	PERS robtarget H40:=[[108.33,-13.47,-153.24],[0.657572,-0.573127,-0.333582,0.357557],[-1,2,-3,0],[9E+09,-23.5,-50.1962,9E+09,9E+09,9E+09]];
	PERS robtarget H41:=[[106.78,-12.3,-180.44],[0.620126,-0.627649,-0.347001,0.317948],[-1,2,-3,0],[9E+09,-23.5,-50.1962,9E+09,9E+09,9E+09]];
	PERS robtarget H42:=[[107.29,-12.09,-209.23],[0.609617,-0.638486,-0.347041,0.316648],[-1,2,-3,0],[9E+09,-22,-50.1961,9E+09,9E+09,9E+09]];
	PERS robtarget H43:=[[151.42,1.00,-178.62],[0.641458,-0.319044,-0.596643,0.361609],[-1,1,-2,0],[9E+09,2.3391E-05,-89.9999,9E+09,9E+09,9E+09]];
	PERS robtarget H44:=[[151.41,-2.81,-181.55],[0.630186,-0.312225,-0.608538,0.367511],[-1,1,-2,0],[9E+09,-4.93563E-05,-90,9E+09,9E+09,9E+09]];
	PERS robtarget H45:=[[146.47,-4.42,-217.18],[0.639919,-0.321987,-0.598345,0.358905],[-1,1,-2,0],[9E+09,-7.78641E-06,-96,9E+09,9E+09,9E+09]];
	PERS robtarget H46:=[[145.71,-4.23,-254.81],[0.639921,-0.322004,-0.598339,0.358897],[-1,1,-2,0],[9E+09,-0.000496233,-90,9E+09,9E+09,9E+09]];
	PERS robtarget H47:=[[140.89,-9.14,-263.21],[0.710194,-0.342001,-0.385873,0.479337],[0,2,-3,0],[9E+09,7.53534E-05,-90.0001,9E+09,9E+09,9E+09]];
	PERS robtarget H48:=[[143.99,-1.12,-261.20],[0.728356,-0.371184,-0.349473,0.45781],[0,2,-3,0],[9E+09,-4.93563E-05,-90,9E+09,9E+09,9E+09]];
    PERS robtarget H49:=[[139.39,0.04,-263.43],[0.692369,-0.514594,-0.306839,0.402081],[0,3,-4,0],[9E+09,0.000594977,-90,9E+09,9E+09,9E+09]];

	PERS robtarget H50:=[[118.68,-79.14,-184.29],[0.585598,-0.475081,0.504836,-0.420137],[-1,1,-2,0],[9E+09,1.99993,81,9E+09,9E+09,9E+09]];
	PERS robtarget H51:=[[100.04,-72.41,-144.62],[0.366328,-0.602136,-0.49492,0.508222],[-1,-2,1,0],[9E+09,-5.97862,-90.0053,9E+09,9E+09,9E+09]];
	PERS robtarget H52:=[[102.34,-25.88,-157.75],[0.366327,-0.602138,-0.494919,0.508222],[-1,-2,1,0],[9E+09,-5.97862,-90.0053,9E+09,9E+09,9E+09]];
	PERS robtarget H53:=[[102.74,-20.19,-159.49],[0.422028,-0.65777,-0.448362,0.433824],[-1,-2,1,0],[9E+09,-5.9786,-90.0052,9E+09,9E+09,9E+09]];
	PERS robtarget H54:=[[120.26,-80.06,-182.83],[0.562619,-0.501182,0.519005,-0.403624],[-1,1,-2,0],[9E+09,3.00001,83.0001,9E+09,9E+09,9E+09]];
	PERS robtarget H55:=[[118.03,-29.06,-194.91],[0.620748,-0.499713,0.456833,-0.395302],[-1,1,-2,0],[9E+09,3.00001,82.9999,9E+09,9E+09,9E+09]];
	PERS robtarget H56:=[[100.61,-21.59,-159.10],[0.506741,-0.624171,-0.339688,0.488095],[-1,-1,1,0],[9E+09,2.59754E-05,-90.0022,9E+09,9E+09,9E+09]];
	PERS robtarget H57:=[[100.74,-23.77,-158.40],[0.460755,-0.573632,-0.396138,0.549296],[-1,-2,1,0],[9E+09,2.59754E-05,-90.0022,9E+09,9E+09,9E+09]];
	PERS robtarget H58:=[[100.20,-73.55,-145.24],[0.453285,-0.563309,-0.404643,0.559893],[-1,-2,1,0],[9E+09,-5.20202E-06,-90.0021,9E+09,9E+09,9E+09]];
    PERS robtarget H59:=[[111.03,-77.81,-189.53],[0.588099,-0.47989,0.482771,-0.436782],[-1,1,-2,0],[9E+09,3.00089,82.9986,9E+09,9E+09,9E+09]];

    PERS robtarget H98:=[[0,0,0],[0.73728,3.31828E-06,0.675588,2.33895E-06],[0,-1,0,0],[9E+09,9E+09,9E+09,9E+09,9E+09,9E+09]];
    PERS robtarget H99:=[[0,0,0],[0.73728,3.31828E-06,0.675588,2.33895E-06],[0,-1,0,0],[9E+09,9E+09,9E+09,9E+09,9E+09,9E+09]];

	PERS robtarget J1:=[[73.79,-16.15,-231.69],[0.592804,-0.401242,-0.200049,-0.669006],[-1,0,-2,0],[9E+09,20.3,-0.000874071,9E+09,9E+09,9E+09]];
	PERS robtarget J2:=[[83.36,-16.67,-232.23],[0.565018,-0.439497,-0.155442,-0.68076],[-1,0,-2,0],[9E+09,20.3,-0.000762002,9E+09,9E+09,9E+09]];
	PERS robtarget J3:=[[70.42,-14.81,-230.39],[0.645916,-0.288855,-0.284725,-0.646751],[-1,0,-2,0],[9E+09,20.3,-0.000874071,9E+09,9E+09,9E+09]];
	PERS robtarget J4:=[[0,-14.81,-230.39],[0.645916,-0.288853,-0.284725,-0.646752],[-1,0,-2,0],[9E+09,20.3,-0.000874071,9E+09,9E+09,9E+09]];
	PERS robtarget J5:=[[0,0,0],[0.73728,3.31828E-06,0.675588,2.33895E-06],[0,-1,0,0],[9E+09,9E+09,9E+09,9E+09,9E+09,9E+09]];

	PERS robtarget K1:=[[-87.2,-16.87,-232.73],[0.672861,-0.201577,-0.388086,-0.596669],[-1,0,-2,0],[9E+09,20.3,-0.000537865,9E+09,9E+09,9E+09]];
	PERS robtarget K2:=[[-95.39,-17.01,-232.66],[0.6898,-0.136714,-0.438311,-0.559793],[-1,0,-3,0],[9E+09,20.3,-0.000649933,9E+09,9E+09,9E+09]];
	PERS robtarget K3:=[[-77.34,-13.76,-231.53],[0.645912,-0.288853,-0.284724,-0.646757],[-1,0,-2,0],[9E+09,20.3,-0.000605106,9E+09,9E+09,9E+09]];
	PERS robtarget K4:=[[0,-13.76,-231.53],[0.645911,-0.288852,-0.284724,-0.646758],[-1,0,-2,0],[9E+09,20.3,-0.000649933,9E+09,9E+09,9E+09]];
	PERS robtarget K5:=[[0,0,0],[0.73728,3.31828E-06,0.675588,2.33895E-06],[0,-1,0,0],[9E+09,9E+09,9E+09,9E+09,9E+09,9E+09]];

	PERS robtarget L1:=[[0,0,0],[0.73728,3.31828E-06,0.675588,2.33895E-06],[0,-1,0,0],[9E+09,9E+09,9E+09,9E+09,9E+09,9E+09]];
	PERS robtarget L2:=[[0,0,0],[0.73728,3.31828E-06,0.675588,2.33895E-06],[0,-1,0,0],[9E+09,9E+09,9E+09,9E+09,9E+09,9E+09]];
	PERS robtarget L3:=[[0,0,0],[0.73728,3.31828E-06,0.675588,2.33895E-06],[0,-1,0,0],[9E+09,9E+09,9E+09,9E+09,9E+09,9E+09]];
	PERS robtarget L4:=[[0,0,0],[0.73728,3.31828E-06,0.675588,2.33895E-06],[0,-1,0,0],[9E+09,9E+09,9E+09,9E+09,9E+09,9E+09]];
    PERS robtarget L5:=[[0,0,0],[0.73728,3.31828E-06,0.675588,2.33895E-06],[0,-1,0,0],[9E+09,9E+09,9E+09,9E+09,9E+09,9E+09]];
    PERS robtarget L6:=[[0,0,0],[0.73728,3.31828E-06,0.675588,2.33895E-06],[0,-1,0,0],[9E+09,9E+09,9E+09,9E+09,9E+09,9E+09]];
    PERS robtarget L7:=[[0,0,0],[0.73728,3.31828E-06,0.675588,2.33895E-06],[0,-1,0,0],[9E+09,9E+09,9E+09,9E+09,9E+09,9E+09]];
    PERS robtarget L8:=[[0,0,0],[0.73728,3.31828E-06,0.675588,2.33895E-06],[0,-1,0,0],[9E+09,9E+09,9E+09,9E+09,9E+09,9E+09]];
    PERS robtarget L9:=[[0,0,0],[0.73728,3.31828E-06,0.675588,2.33895E-06],[0,-1,0,0],[9E+09,9E+09,9E+09,9E+09,9E+09,9E+09]];
    PERS robtarget L10:=[[0,0,0],[0.73728,3.31828E-06,0.675588,2.33895E-06],[0,-1,0,0],[9E+09,9E+09,9E+09,9E+09,9E+09,9E+09]];
    PERS robtarget L40:=[[0,-169.39,841.37],[0.442606,-0.811905,0.276598,-0.261544],[-1,1,-2,0],[9E+09,-14.1988,49.3012,9E+09,9E+09,9E+09]];
	PERS robtarget L41:=[[96.6934,-167.187,469.006],[0.634627,-0.665497,0.280508,-0.275094],[0,1,-2,0],[9E+09,-0.275255,46.2247,9E+09,9E+09,9E+09]];
	PERS robtarget L42:=[[96.95,-163.039,524.102],[0.613381,-0.680757,0.277205,-0.288948],[-1,1,-2,0],[9E+09,-3.95049,47.5495,9E+09,9E+09,9E+09]];
	PERS robtarget L43:=[[96.4403,0,0],[0.73728,3.31828E-06,0.675588,2.33895E-06],[0,-1,0,0],[9E+09,9E+09,9E+09,9E+09,9E+09,9E+09]];
	PERS robtarget L44:=[[96.4403,0,0],[0.73728,3.31828E-06,0.675588,2.33895E-06],[0,-1,0,0],[9E+09,9E+09,9E+09,9E+09,9E+09,9E+09]];
    PERS robtarget L45:=[[97.2063,-156.283,579.142],[0.580686,-0.706216,0.267929,-0.303771],[-1,1,-2,0],[9E+09,-8.10884,48.3912,9E+09,9E+09,9E+09]];
    PERS robtarget L46:=[[97.2552,-152.576,589.64],[0.574791,-0.71088,0.269371,-0.302828],[-1,1,-2,0],[9E+09,-8.96447,48.5355,9E+09,9E+09,9E+09]];
    PERS robtarget L47:=[[97.4579,-143.314,633.167],[0.544782,-0.734855,0.260153,-0.309065],[-1,1,-2,0],[9E+09,-12.438,49.062,9E+09,9E+09,9E+09]];
    PERS robtarget L48:=[[97.7028,-125.721,685.736],[0.505031,-0.765566,0.242802,-0.31607],[-1,1,-2,0],[9E+09,-16.8632,49.6368,9E+09,9E+09,9E+09]];
    PERS robtarget L49:=[[97.7897,-118.231,704.402],[0.49199,-0.775329,0.234663,-0.318974],[-1,1,-2,0],[9E+09,-18.2042,49.7958,9E+09,9E+09,9E+09]];
    PERS robtarget L50:=[[97.7897,-112.37,718.21],[0.610407,-0.715463,0.144537,-0.307611],[-1,1,-3,0],[9E+09,-18.2042,49.7958,9E+09,9E+09,9E+09]];

    PERS robtarget L40cramp1:=[[89.34,-171.59,828.86],[0.371994,-0.853426,0.291056,-0.220391],[-1,1,-2,0],[9E+09,-14.1988,49.3012,9E+09,9E+09,9E+09]];
    PERS robtarget L40cramp2:=[[89.66,-174.94,816.24],[0.319922,-0.878441,0.2998,-0.19003],[-1,1,-2,0],[9E+09,-14.1988,49.3012,9E+09,9E+09,9E+09]];


    PERS robtarget L68:=[[96.3294,-183.624,325.052],[0.732807,-0.547572,0.316136,-0.25143],[0,2,-3,0],[9E+09,11.563,48.937,9E+09,9E+09,9E+09]];
    PERS robtarget L69:=[[96.3488,-150.2,298.164],[0.659613,-0.633434,0.346072,-0.20954],[0,2,-2,0],[9E+09,9.82577,48.6742,9E+09,9E+09,9E+09]];
    PERS robtarget L67:=[[96.3401,-153.031,310.32],[0.720285,-0.563292,0.323715,-0.243106],[0,2,-3,0],[9E+09,8.96447,48.5355,9E+09,9E+09,9E+09]];
    PERS robtarget L66:=[[96.3373,-176.27,314.16],[0.672496,-0.593746,0.194944,-0.396502],[0,1,-3,0],[9E+09,11.0978,49.3364,9E+09,9E+09,9E+09]];
    PERS robtarget L65:=[[96.3969,-150.45,231.45],[0.672501,-0.59375,0.194937,-0.39649],[0,1,-2,0],[9E+09,15.8071,49.3364,9E+09,9E+09,9E+09]];
    PERS robtarget L64:=[[96.3969,-150.45,231.45],[0.672501,-0.59375,0.194937,-0.39649],[0,1,-2,0],[9E+09,15.8071,49.3364,9E+09,9E+09,9E+09]];
    PERS robtarget L63:=[[96.3115,-190.14,349.956],[0.72386,-0.558889,0.31987,-0.247696],[0,2,-3,0],[9E+09,9.82577,48.6742,9E+09,9E+09,9E+09]];
    PERS robtarget L62:=[[96.3013,-197.227,383.785],[0.712549,-0.57296,0.323832,-0.243152],[0,2,-3,0],[9E+09,7.68338,48.3166,9E+09,9E+09,9E+09]];
    PERS robtarget L61:=[[96.3326,-155.291,320.651],[0.74323,-0.532709,0.302829,-0.268562],[0,2,-3,0],[9E+09,8.10884,48.3912,9E+09,9E+09,9E+09]];
    PERS robtarget L60:=[[0,-199.67,711.03],[0.694049,-0.59574,0.215139,-0.342208],[-1,2,-3,0],[9E+09,-6.41779,48.0822,9E+09,9E+09,9E+09]];

	PERS robtarget M70:=[[-93.6428,-146.142,278.519],[0.617494,-0.211758,-0.675695,-0.342485],[-1,0,-2,0],[9E+09,9.82577,-48.6742,9E+09,9E+09,9E+09]];
	PERS robtarget L70:=[[96.3488,-145.531,278.717],[0.5807,-0.736812,0.322963,-0.124864],[0,2,-2,0],[9E+09,9.82577,48.6742,9E+09,9E+09,9E+09]];

    PERS robtarget M69:=[[-93.6428,-150.811,297.966],[0.566281,-0.122383,-0.698677,-0.419761],[-1,0,-2,0],[9E+09,9.82577,-48.6742,9E+09,9E+09,9E+09]];
    PERS robtarget M68:=[[-93.4449,-183.819,325.057],[0.649099,-0.0877175,-0.626165,-0.422957],[-1,0,-2,0],[9E+09,11.563,-48.937,9E+09,9E+09,9E+09]];
    PERS robtarget M67:=[[-93.5531,-153.581,310.245],[0.640867,-0.100792,-0.641818,-0.408901],[-1,0,-2,0],[9E+09,8.96447,-48.5355,9E+09,9E+09,9E+09]];
    PERS robtarget M66:=[[-93.5299,-177.55,313.42],[0.638045,-0.136384,-0.644614,-0.398463],[-1,0,-2,0],[9E+09,7.72271,-42.4887,9E+09,9E+09,9E+09]];
    PERS robtarget M65:=[[-94.1287,-400.46,231.46],[0.672498,-0.593754,0.194941,-0.396487],[0,1,-2,0],[9E+09,15.8062,49.3364,9E+09,9E+09,9E+09]];
    PERS robtarget M64:=[[-94.1287,-400.46,231.46],[0.672498,-0.593754,0.194941,-0.396487],[0,1,-2,0],[9E+09,15.8062,49.3364,9E+09,9E+09,9E+09]];
    PERS robtarget M63:=[[-93.2634,-190.289,349.9],[0.657211,-0.117717,-0.633101,-0.391663],[-1,0,-2,0],[9E+09,9.82577,-48.6742,9E+09,9E+09,9E+09]];
    PERS robtarget M62:=[[-93.0156,-197.372,383.803],[0.666771,-0.159333,-0.638564,-0.349665],[-1,0,-2,0],[9E+09,7.68338,-48.3166,9E+09,9E+09,9E+09]];
    PERS robtarget M61:=[[-93.4777,-155.55,320.558],[0.705794,-0.145598,-0.601393,-0.34494],[-1,0,-2,0],[9E+09,8.10884,-48.3912,9E+09,9E+09,9E+09]];
    PERS robtarget M60:=[[0,-199.66,711.57],[0.723621,-0.258575,-0.586981,-0.254884],[-1,0,-2,0],[9E+09,-6.41779,-48.0822,9E+09,9E+09,9E+09]];

	PERS robtarget M1:=[[0,0,0],[0.73728,3.31828E-06,0.675588,2.33895E-06],[0,-1,0,0],[9E+09,9E+09,9E+09,9E+09,9E+09,9E+09]];
	PERS robtarget M2:=[[0,0,0],[0.73728,3.31828E-06,0.675588,2.33895E-06],[0,-1,0,0],[9E+09,9E+09,9E+09,9E+09,9E+09,9E+09]];
	PERS robtarget M3:=[[0,0,0],[0.73728,3.31828E-06,0.675588,2.33895E-06],[0,-1,0,0],[9E+09,9E+09,9E+09,9E+09,9E+09,9E+09]];
	PERS robtarget M4:=[[0,0,0],[0.73728,3.31828E-06,0.675588,2.33895E-06],[0,-1,0,0],[9E+09,9E+09,9E+09,9E+09,9E+09,9E+09]];
    PERS robtarget M5:=[[0,0,0],[0.73728,3.31828E-06,0.675588,2.33895E-06],[0,-1,0,0],[9E+09,9E+09,9E+09,9E+09,9E+09,9E+09]];
    PERS robtarget M6:=[[0,0,0],[0.73728,3.31828E-06,0.675588,2.33895E-06],[0,-1,0,0],[9E+09,9E+09,9E+09,9E+09,9E+09,9E+09]];
    PERS robtarget M7:=[[0,0,0],[0.73728,3.31828E-06,0.675588,2.33895E-06],[0,-1,0,0],[9E+09,9E+09,9E+09,9E+09,9E+09,9E+09]];
    PERS robtarget M8:=[[0,0,0],[0.73728,3.31828E-06,0.675588,2.33895E-06],[0,-1,0,0],[9E+09,9E+09,9E+09,9E+09,9E+09,9E+09]];
    PERS robtarget M9:=[[0,0,0],[0.73728,3.31828E-06,0.675588,2.33895E-06],[0,-1,0,0],[9E+09,9E+09,9E+09,9E+09,9E+09,9E+09]];
    PERS robtarget M10:=[[111.15,-112.53,220.41],[0.643491,-0.632415,0.208259,-0.377624],[0,1,-2,0],[9E+09,10.5848,49.3365,9E+09,9E+09,9E+09]];
    PERS robtarget M40:=[[0,-168.58,841.23],[0.497618,-0.44465,-0.735594,-0.116468],[-1,0,-2,0],[9E+09,-14.1988,-49.3012,9E+09,9E+09,9E+09]];
	PERS robtarget M41:=[[-92.3859,-167.501,469.014],[0.646009,-0.277625,-0.665978,-0.249139],[-1,0,-2,0],[9E+09,-0.275255,-46.2247,9E+09,9E+09,9E+09]];
	PERS robtarget M42:=[[-92.0275,-163.382,524.16],[0.641706,-0.296382,-0.672629,-0.218956],[-1,0,-2,0],[9E+09,-3.95049,-47.5495,9E+09,9E+09,9E+09]];
	PERS robtarget M43:=[[-95.7201,0,0],[0.73728,3.31828E-06,0.675588,2.33895E-06],[0,-1,0,0],[9E+09,9E+09,9E+09,9E+09,9E+09,9E+09]];
	PERS robtarget M44:=[[-95.7201,0,0],[0.73728,3.31828E-06,0.675588,2.33895E-06],[0,-1,0,0],[9E+09,9E+09,9E+09,9E+09,9E+09,9E+09]];
    PERS robtarget M45:=[[-92.0423,-156.01,579.07],[0.629623,-0.325223,-0.681731,-0.181791],[-1,0,-2,0],[9E+09,-8.10884,-48.3912,9E+09,9E+09,9E+09]];
    PERS robtarget M46:=[[-92.0451,-152.729,589.619],[0.622938,-0.320879,-0.689165,-0.184493],[-1,0,-2,0],[9E+09,-8.96447,-48.5355,9E+09,9E+09,9E+09]];
    PERS robtarget M47:=[[-92.0568,-142.72,632.959],[0.608305,-0.355764,-0.693631,-0.149241],[-1,0,-2,0],[9E+09,-12.438,-49.062,9E+09,9E+09,9E+09]];
    PERS robtarget M48:=[[-92.0709,-124.754,685.369],[0.582927,-0.382483,-0.706223,-0.123094],[-1,0,-2,0],[9E+09,-16.8632,-49.6368,9E+09,9E+09,9E+09]];
    PERS robtarget M49:=[[-92.0759,-117.236,703.903],[0.574484,-0.388531,-0.710806,-0.117328],[-1,0,-2,0],[9E+09,-18.2042,-49.7958,9E+09,9E+09,9E+09]];
    PERS robtarget M50:=[[-92.0759,-111.375,717.71],[0.628488,-0.31192,-0.682674,-0.204122],[-1,0,-2,0],[9E+09,-18.2042,-49.7958,9E+09,9E+09,9E+09]];


!!!!!!!!!!!!!!!!!!!!!!END OF THE WRAPPER WELDS!!!!!!!!!!

	PERS robtarget AIRG50_1:=[[-520.73,-53.52,-86.29],[0.528398,-0.491715,0.591821,-0.358833],[-1,-3,2,0],[9E+09,-5.99999,96.0001,9E+09,9E+09,9E+09]];
	CONST robtarget AIRTOG40:=[[-143.55,-8.66,-258.80],[0.531165,-0.426072,0.558082,-0.474208],[-1,1,-2,0],[9E+09,4.25678,88.0425,9E+09,9E+09,9E+09]];
	CONST robtarget AIRTOG50:=[[-113.36,-82.97,-180.83],[0.229441,0.62405,-0.35786,-0.655634],[-1,-1,-3,0],[9E+09,2,-81,9E+09,9E+09,9E+09]];
	CONST robtarget AIRTOH50:=[[115.64,-84.86,-185.39],[0.583759,-0.477077,0.502947,-0.422693],[-1,1,-2,0],[9E+09,1.99998,81,9E+09,9E+09,9E+09]];
	CONST robtarget AIRTOH40:=[[147.28,-7.36,-258.56],[0.639947,-0.321989,-0.598323,0.35889],[-1,1,-2,0],[9E+09,0.0012601,-90,9E+09,9E+09,9E+09]];
	CONST robtarget AIRTOSNIFF_FRONT1:=[[-32.84,651.47,382.08],[0.458666,0.489208,0.507975,0.540615],[0,0,-2,1],[9E+09,0.00155109,179.999,9E+09,9E+09,9E+09]];
	CONST robtarget AIRTOSNIFF_FRONT2:=[[65.52,66.66,373.83],[0.458667,0.489243,0.508101,0.540464],[0,0,-2,1],[9E+09,0.00077165,180,9E+09,9E+09,9E+09]];
	CONST robtarget AIRTOSNIFF_BACK1:=[[30.52,-723.52,526.87],[0.502022,0.5218,-0.484293,-0.491081],[-1,-1,-2,1],[9E+09,0,0,9E+09,9E+09,9E+09]];


	CONST robtarget AIRTOU30_1:=[[288.8,655.25,389.82],[0.299157,-0.329043,-0.63518,0.631493],[-1,1,-2,0],[9E+09,-22,-135,9E+09,9E+09,9E+09]];
    CONST robtarget SPAGHAIR1:=[[10.28,-310.74,36.91],[0.687984,-0.0566141,-0.0392933,-0.722448],[0,-1,-1,0],[9E+09,0.000407913,0.000403513,9E+09,9E+09,9E+09]];
    CONST robtarget SPAGHAIR2:=[[6.27,-351.73,67.88],[0.547219,-0.440868,-0.452479,-0.549046],[-1,0,-2,0],[9E+09,0.000906752,0.000784547,9E+09,9E+09,9E+09]];
    CONST robtarget SPAGHAIR3:=[[-0.30,-21.47,198.76],[0.547881,-0.439991,-0.453355,-0.548365],[-1,0,-2,0],[9E+09,0.000927537,0.000829375,9E+09,9E+09,9E+09]];
    CONST robtarget SPAGHAIRp180:=[[0.12,-168.40,-471.89],[0.525941,0.414544,0.456451,-0.585828],[0,0,-4,0],[9E+09,-0.00069369,180,9E+09,9E+09,9E+09]];
    CONST robtarget AIRTOT30_1:=[[-387.74,-383.85,499.37],[0.413094,-0.652879,0.573252,-0.27292],[0,2,-3,0],[9E+09,-18.7937,76.4339,9E+09,9E+09,9E+09]];
    CONST robtarget AIRTOT30_2:=[[-149.56,-360.66,399.66],[0.413095,-0.652876,0.573254,-0.272923],[0,2,-2,0],[9E+09,-18.7937,76.4339,9E+09,9E+09,9E+09]];
    CONST robtarget AIRTOHSIDESEARCH_1:=[[336.07,-164.67,-442.68],[0.254905,-0.945405,0.203005,0.00489991],[-1,1,-1,0],[9E+09,0.000127316,-4.4762E-05,9E+09,9E+09,9E+09]];
    CONST robtarget AIRTOGSIDESEARCH_1:=[[-336.31,363.60,-301.34],[0.0476339,-0.197008,-0.979243,0.00193439],[-1,1,-1,0],[9E+09,0.0487537,179.953,9E+09,9E+09,9E+09]];

    CONST robtarget AIRTOU30_2:=[[-69.31,237.05,289.11],[0.401333,0.727401,-0.0339958,0.555577],[-1,0,-2,0],[9E+09,-22,-225,9E+09,9E+09,9E+09]];
    CONST robtarget AIRTOT30_3:=[[399.86,-369.93,558.91],[0.724495,0.0577651,-0.674607,0.129141],[-1,0,-2,0],[9E+09,-10.5388,-76.9656,9E+09,9E+09,9E+09]];
    CONST robtarget AIRTOAH118:=[[414.86,-318.11,504.4],[0.600973,-0.149246,-0.783454,-0.0525223],[-1,0,-2,0],[9E+09,-40,-74.7502,9E+09,9E+09,9E+09]];
    CONST robtarget AIRTOAG118:=[[-319.97,-306.98,657.22],[0.263609,-0.69609,0.660491,-0.098598],[-1,0,-1,0],[9E+09,-40,100,9E+09,9E+09,9E+09]];
    CONST robtarget AIRTOAH119:=[[-78.91,-59.71,-33.25],[0.0723101,-0.842822,0.383137,0.370983],[0,3,-3,0],[9E+09,-42,-76.0788,9E+09,9E+09,9E+09]];
    CONST robtarget AIRTOAH120:=[[528.62,-833.93,882.62],[0.0951167,0.895249,0.241984,-0.361838],[0,3,-3,0],[9E+09,-40,-90,9E+09,9E+09,9E+09]];

    PERS robtarget AIRH50_1:=[[387.44,-242.61,-609.79],[0.430453,-0.560647,-0.430883,0.561004],[0,-1,1,0],[9E+09,-7.78641E-06,-90,9E+09,9E+09,9E+09]];

    PERS robtarget AIRTOJKSEARCH:=[[13.2,-349.36,-242.95],[0.0768042,0.297355,-0.535013,-0.787047],[-1,0,-3,0],[9E+09,20.3,0.000170104,9E+09,9E+09,9E+09]];
    PERS robtarget AIRTOJKSEARCH2:=[[8.75,-307.76,-107.1],[0.724947,-0.0658517,-0.0586667,-0.683136],[-1,0,-2,0],[9E+09,9.5,0.000403513,9E+09,9E+09,9E+09]];
    PERS robtarget AIRTOJK:=[[-12.97,-407.01,-486.33],[0.666181,-0.303759,-0.293409,-0.61469],[-1,0,-2,0],[9E+09,20.3,0,9E+09,9E+09,9E+09]];


    PERS robtarget P1:=[[101.57,-24.25,201.66],[0.0129324,-0.0134658,-0.680078,0.732902],[0,2,-3,0],[9E+09,-18.5,180,9E+09,9E+09,9E+09]];
    PERS robtarget P2:=[[19.22,-24.62,201.94],[0.00205672,-0.00263914,0.680199,-0.73302],[0,2,-3,0],[9E+09,-18.5,180,9E+09,9E+09,9E+09]];
    PERS robtarget P1E:=[[59.01,-25.54,202.44],[0.0129283,-0.0134686,-0.680079,0.732901],[0,2,-3,0],[9E+09,-18.5,180,9E+09,9E+09,9E+09]];
    PERS robtarget P2E:=[[68.01,-25.07,202.62],[0.00204531,-0.00263582,0.680198,-0.733021],[0,2,-3,0],[9E+09,-18.5,180,9E+09,9E+09,9E+09]];
    PERS robtarget P3:=[[0,0,0],[0.73728,3.31828E-06,0.675588,2.33895E-06],[0,-1,0,0],[9E+09,9E+09,9E+09,9E+09,9E+09,9E+09]];
    PERS robtarget P4:=[[0,0,0],[0.73728,3.31828E-06,0.675588,2.33895E-06],[0,-1,0,0],[9E+09,9E+09,9E+09,9E+09,9E+09,9E+09]];
    PERS robtarget P11:=[[-32.11,310.00,277.38],[0.229339,0.33529,-0.673696,0.617348],[-1,1,-2,0],[9E+09,-31.4536,167.903,9E+09,9E+09,9E+09]];
    PERS robtarget P12:=[[0,0,0],[0.73728,3.31828E-06,0.675588,2.33895E-06],[0,-1,0,0],[9E+09,9E+09,9E+09,9E+09,9E+09,9E+09]];
    PERS robtarget P11E:=[[-32.10,310.00,277.38],[0.22934,0.335293,-0.673695,0.617348],[-1,1,-2,0],[9E+09,-31.4536,167.903,9E+09,9E+09,9E+09]];
    PERS robtarget P12E:=[[0,0,0],[0.73728,3.31828E-06,0.675588,2.33895E-06],[0,-1,0,0],[9E+09,9E+09,9E+09,9E+09,9E+09,9E+09]];


    PERS robtarget Q1:=[[-104.68,-25.08,202.31],[0.00202495,-0.00263121,0.680193,-0.733025],[0,2,-2,0],[9E+09,-18.5,180,9E+09,9E+09,9E+09]];
    PERS robtarget Q2:=[[-23.01,-24.18,202.57],[0.0125721,-0.0130962,-0.680083,0.732911],[0,2,-3,0],[9E+09,-18.5,180,9E+09,9E+09,9E+09]];
    PERS robtarget Q1E:=[[-59.01,-26.25,202.30],[0.00202647,-0.00263226,0.680194,-0.733024],[0,2,-3,0],[9E+09,-18.5,180,9E+09,9E+09,9E+09]];
    PERS robtarget Q2E:=[[-67.98,-25.79,202.24],[0.0125711,-0.0130979,-0.680081,0.732912],[0,2,-3,0],[9E+09,-18.5,180,9E+09,9E+09,9E+09]];
    PERS robtarget Q3:=[[0,0,0],[0.73728,3.31828E-06,0.675588,2.33895E-06],[0,-1,0,0],[9E+09,9E+09,9E+09,9E+09,9E+09,9E+09]];
    PERS robtarget Q4:=[[0,0,0],[0.73728,3.31828E-06,0.675588,2.33895E-06],[0,-1,0,0],[9E+09,9E+09,9E+09,9E+09,9E+09,9E+09]];
    PERS robtarget Q11:=[[-32.11,310.00,277.38],[0.22934,0.335291,-0.673695,0.617348],[-1,1,-2,0],[9E+09,-31.4535,167.903,9E+09,9E+09,9E+09]];
    PERS robtarget Q12:=[[0,0,0],[0.73728,3.31828E-06,0.675588,2.33895E-06],[0,-1,0,0],[9E+09,9E+09,9E+09,9E+09,9E+09,9E+09]];
    PERS robtarget Q11E:=[[-32.11,310.00,277.38],[0.22934,0.335291,-0.673695,0.617348],[-1,1,-2,0],[9E+09,-31.4536,167.903,9E+09,9E+09,9E+09]];
    PERS robtarget Q12E:=[[0,0,0],[0.73728,3.31828E-06,0.675588,2.33895E-06],[0,-1,0,0],[9E+09,9E+09,9E+09,9E+09,9E+09,9E+09]];

    PERS robtarget R1:=[[-96.76,-3.06,-203.38],[0.00343762,-0.00492383,-0.780506,0.625119],[-1,1,-2,0],[9E+09,24.5,180,9E+09,9E+09,9E+09]];
    PERS robtarget R2:=[[96.76,-3.06,-203.38],[0.00343762,-0.00492383,-0.780506,0.625119],[-1,1,-2,0],[9E+09,24.5,180,9E+09,9E+09,9E+09]];
    PERS robtarget R5:=[[-104.69,-2.72,-204.58],[0.00094552,-0.000652264,0.713871,-0.700276],[-1,1,-2,0],[9E+09,24.5,180,9E+09,9E+09,9E+09]];
    PERS robtarget R6:=[[0,-2.72,-204.58],[0.00094552,-0.000652264,0.713871,-0.700276],[-1,1,-2,0],[9E+09,24.5,180,9E+09,9E+09,9E+09]];
    PERS robtarget S1:=[[0,0,0],[0.73728,3.31828E-06,0.675588,2.33895E-06],[0,-1,0,0],[9E+09,9E+09,9E+09,9E+09,9E+09,9E+09]];
    PERS robtarget S2:=[[0,0,0],[0.73728,3.31828E-06,0.675588,2.33895E-06],[0,-1,0,0],[9E+09,9E+09,9E+09,9E+09,9E+09,9E+09]];
    PERS robtarget S5:=[[104.69,-2.72,-204.58],[0.00094552,-0.000652264,0.713871,-0.700276],[-1,1,-2,0],[9E+09,24.5,180,9E+09,9E+09,9E+09]];
    PERS robtarget S6:=[[-8,-2.72,-204.58],[0.00094552,-0.000652264,0.713871,-0.700276],[-1,1,-2,0],[9E+09,24.5,180,9E+09,9E+09,9E+09]];

    PERS robtarget T1:=[[95.95,-65.01,159.52],[0.641802,-0.422701,-0.339875,-0.542125],[-1,0,-2,0],[9E+09,41,0.000982197,9E+09,9E+09,9E+09]];
    PERS robtarget T2:=[[0,0,0],[0.73728,3.31828E-06,0.675588,2.33895E-06],[0,-1,0,0],[9E+09,9E+09,9E+09,9E+09,9E+09,9E+09]];
    PERS robtarget T11:=[[103.36,-64.34,159.29],[0.6272,-0.444915,-0.366585,-0.523724],[-1,0,-2,0],[9E+09,38,0.000332198,9E+09,9E+09,9E+09]];
    PERS robtarget T12:=[[0,-64.34,159.29],[0.6272,-0.444915,-0.366585,-0.523724],[-1,0,-2,0],[9E+09,38,0.000332198,9E+09,9E+09,9E+09]];
    PERS robtarget T20:=[[0,0,0],[0.73728,3.31828E-06,0.675588,2.33895E-06],[0,-1,0,0],[9E+09,-13.4,9E+09,9E+09,9E+09,9E+09]];
    PERS robtarget T21:=[[16.06,-32.26,244.00],[0.455639,-0.889634,-0.00344562,-0.0305311],[0,2,-2,0],[9E+09,-13.4,0.000690818,9E+09,9E+09,9E+09]];
    PERS robtarget T22:=[[39.41,-32.23,244.11],[0.412338,-0.909307,0.0129589,-0.0545063],[0,2,-2,0],[9E+09,-13.4,0.000578749,9E+09,9E+09,9E+09]];

    PERS robtarget U1:=[[-95.95,-65.02,159.54],[0.641805,-0.422704,-0.339872,-0.54212],[-1,0,-2,0],[9E+09,41,0.00109427,9E+09,9E+09,9E+09]];
    PERS robtarget U2:=[[0,0,0],[0.73728,3.31828E-06,0.675588,2.33895E-06],[0,-1,0,0],[9E+09,9E+09,9E+09,9E+09,9E+09,9E+09]];
    PERS robtarget U11:=[[-104.63,-64.64,160.25],[0.627203,-0.444915,-0.366586,-0.523719],[-1,0,-2,0],[9E+09,38,0.00028737,9E+09,9E+09,9E+09]];
    PERS robtarget U12:=[[10.00,-64.69,160.46],[0.6272,-0.444913,-0.366584,-0.523726],[-1,0,-2,0],[9E+09,38,0.000332198,9E+09,9E+09,9E+09]];
    PERS robtarget U20:=[[0,0,0],[0.73728,3.31828E-06,0.675588,2.33895E-06],[0,-1,0,0],[9E+09,-13.4,9E+09,9E+09,9E+09,9E+09]];
    PERS robtarget U21:=[[-16.39,-34.08,245.33],[0.461761,-0.885885,-0.0346826,0.0279648],[0,2,-3,0],[9E+09,-13.4,0.00064599,9E+09,9E+09,9E+09]];
    PERS robtarget U22:=[[-44.48,-34.20,245.31],[0.417737,-0.906887,-0.0400182,0.0380858],[0,2,-2,0],[9E+09,-13.4,0.00064599,9E+09,9E+09,9E+09]];

    PERS robtarget T30:=[[90.88,-54.85,307.26],[0.450858,-0.712146,0.523746,-0.123556],[0,2,-2,0],[9E+09,-30.0001,62.5001,9E+09,9E+09,9E+09]];
    PERS robtarget T31:=[[91.58,-38.24,311.00],[0.51439,-0.645709,0.560108,-0.0688631],[0,2,-2,0],[9E+09,-35,75.0002,9E+09,9E+09,9E+09]];
    PERS robtarget T32:=[[90.24,-72.06,303.57],[0.365292,-0.71172,0.572567,-0.179396],[0,2,-3,0],[9E+09,-30,50,9E+09,9E+09,9E+09]];
    PERS robtarget T33:=[[91.65,-73.78,297.92],[0.313537,-0.654642,-0.246837,-0.642036],[-1,1,-2,0],[9E+09,16,44.9999,9E+09,9E+09,9E+09]];
    PERS robtarget T34:=[[90.87,-68.13,246.36],[0.328379,-0.641609,-0.258328,-0.643251],[-1,1,-2,0],[9E+09,16,45,9E+09,9E+09,9E+09]];
    PERS robtarget T35:=[[91.55,-67.45,235.06],[0.32294,-0.723435,-0.31569,-0.522198],[-1,1,-2,0],[9E+09,16,45.0001,9E+09,9E+09,9E+09]];
    PERS robtarget T36:=[[93.34,-32.21,301.41],[0.574248,0.712233,0.00342477,0.403672],[-1,0,-2,0],[9E+09,-10,-210,9E+09,9E+09,9E+09]];
    PERS robtarget T37:=[[92.72,-35.19,262.68],[0.530151,0.732682,0.0420282,0.424677],[-1,0,-2,0],[9E+09,-14,-225,9E+09,9E+09,9E+09]];
    PERS robtarget T38:=[[90.91,-36.56,245.76],[0.498467,0.772759,-0.0129197,0.392692],[-1,0,-2,0],[9E+09,-14,-225,9E+09,9E+09,9E+09]];
    PERS robtarget T39:=[[0,0,0],[0.73728,3.31828E-06,0.675588,2.33895E-06],[0,-1,0,0],[9E+09,9E+09,9E+09,9E+09,9E+09,9E+09]];


    PERS robtarget T40:=[[252.65,-224.59,297.64],[0.447189,-0.874652,-0.149854,-0.112032],[0,1,-2,0],[9E+09,-13.2528,0.000179376,9E+09,9E+09,9E+09]];
    PERS robtarget T41:=[[108.09,-64.72,228.69],[0.636614,-0.377124,-0.488778,0.462165],[0,1,-2,0],[9E+09,1.13325,-89.2762,9E+09,9E+09,9E+09]];
    PERS robtarget T42:=[[104.82,-37.55,237.59],[0.555581,-0.303081,-0.579231,0.513773],[0,1,-3,0],[9E+09,1.13378,-89.2771,9E+09,9E+09,9E+09]];
    PERS robtarget T43:=[[106.68,-36.43,238.40],[0.528442,-0.356066,-0.59819,0.485937],[0,1,-2,0],[9E+09,1.13371,-89.2772,9E+09,9E+09,9E+09]];
	PERS robtarget T44:=[[107.16,-63.22,229.16],[0.600027,-0.429261,-0.523045,0.426764],[0,1,-2,0],[9E+09,1.13366,-89.277,9E+09,9E+09,9E+09]];

    PERS robtarget T50:=[[-104.71,-64.29,229.91],[0.651048,-0.411829,0.470927,-0.429838],[0,2,-3,0],[9E+09,1.01675,89.5592,9E+09,9E+09,9E+09]];
    PERS robtarget T51:=[[-104.84,-38.43,237.08],[0.582543,-0.3488,0.547609,-0.488985],[0,3,-3,0],[9E+09,1.01673,89.5592,9E+09,9E+09,9E+09]];
    PERS robtarget T52:=[[-105.08,-36.51,237.36],[0.540988,-0.355408,0.595162,-0.476234],[0,2,-3,0],[9E+09,1.01667,89.5592,9E+09,9E+09,9E+09]];
    PERS robtarget T53:=[[-106.69,-63.23,230.03],[0.633928,-0.442285,0.493241,-0.39904],[0,2,-3,0],[9E+09,1.01669,89.5595,9E+09,9E+09,9E+09]];
    PERS robtarget T54:=[[-137.13,-21.49,129.92],[0.2715,-0.629431,0.285247,-0.669881],[0,1,-2,0],[9E+09,1.01926,89.5581,9E+09,9E+09,9E+09]];


    PERS robtarget U30:=[[-92.47,-54.63,307.68],[0.0293299,-0.754001,0.453719,0.47409],[0,3,-3,0],[9E+09,-30,-62.5001,9E+09,9E+09,9E+09]];
    PERS robtarget U31:=[[-91.42,-37.33,313.87],[0.0599243,-0.744432,0.395177,0.534851],[0,3,-3,0],[9E+09,-35,-75.0001,9E+09,9E+09,9E+09]];
    PERS robtarget U32:=[[-92.38,-75.31,304.77],[0.00570906,0.770695,-0.444861,-0.456174],[0,3,-3,0],[9E+09,-30,-49.9998,9E+09,9E+09,9E+09]];


    PERS robtarget U33:=[[-93.98,-72.84,296.4],[0.630482,-0.229885,-0.674636,-0.307426],[-1,0,-2,0],[9E+09,16,-45.0001,9E+09,9E+09,9E+09]];
    PERS robtarget U34:=[[-93.26,-67.32,246.12],[0.634948,-0.237327,-0.662121,-0.319551],[-1,0,-2,0],[9E+09,16,-44.9999,9E+09,9E+09,9E+09]];
    PERS robtarget U35:=[[-93.56,-66.31,235.89],[0.558547,-0.302047,-0.705587,-0.314547],[-1,0,-2,0],[9E+09,16,-45,9E+09,9E+09,9E+09]];
    PERS robtarget U36:=[[-97.14,-29.36,301.69],[0.193501,-0.275612,-0.665286,0.666326],[0,1,-2,0],[9E+09,-10,-150,9E+09,9E+09,9E+09]];
    PERS robtarget U37:=[[-96.35,-35.40,263.41],[0.179331,-0.261415,-0.669241,0.672026],[0,1,-2,0],[9E+09,-14,-135,9E+09,9E+09,9E+09]];
    PERS robtarget U38:=[[-93.20,-36.61,245.32],[0.125384,-0.267907,-0.761573,0.576638],[0,1,-2,0],[9E+09,-14,-135,9E+09,9E+09,9E+09]];
    PERS robtarget U39:=[[0,0,0],[0.73728,3.31828E-06,0.675588,2.33895E-06],[0,-1,0,0],[9E+09,9E+09,9E+09,9E+09,9E+09,9E+09]];

    PERS robtarget T70:=[[52.38,-28.30,307.55],[0.456141,-0.209042,-0.69521,-0.514704],[0,0,-2,0],[9E+09,1.24994,-22,9E+09,9E+09,9E+09]];
    PERS robtarget T71:=[[53.53,-23.67,332.89],[0.503214,-0.187589,-0.590415,-0.602492],[0,0,-2,0],[9E+09,1.25001,-22,9E+09,9E+09,9E+09]];
    PERS robtarget T72:=[[-84.29,-45.38,314.72],[0.441867,0.0418055,-0.822139,-0.356504],[0,0,-2,0],[9E+09,-24.6237,-70.4231,9E+09,9E+09,9E+09]];
    PERS robtarget T73:=[[-87.46,-79.02,295.66],[0.66022,-0.251573,-0.673606,-0.216976],[-1,0,-2,0],[9E+09,15.9985,-48.8794,9E+09,9E+09,9E+09]];
    PERS robtarget T74:=[[-86.41,-74.16,254.74],[0.653179,-0.269346,-0.66748,-0.235121],[-1,0,-2,0],[9E+09,15.9986,-48.8795,9E+09,9E+09,9E+09]];
    PERS robtarget T75:=[[-87.75,-71.78,236.69],[0.629807,-0.320201,-0.646779,-0.287215],[-1,0,-2,0],[9E+09,15.9985,-48.8795,9E+09,9E+09,9E+09]];
    PERS robtarget T76:=[[-89.49,-33.65,303.7],[0.231731,-0.261825,-0.662764,0.662189],[0,1,-2,0],[9E+09,-10.7,-142.001,9E+09,9E+09,9E+09]];
    PERS robtarget T77:=[[-87.55,-38.98,264.17],[0.231738,-0.261829,-0.662763,0.662186],[0,1,-2,0],[9E+09,-10.7,-132.001,9E+09,9E+09,9E+09]];
    PERS robtarget T78:=[[-84.41,-40.22,244.47],[0.18148,-0.28897,-0.760586,0.552333],[0,1,-2,0],[9E+09,-10.7,-132.001,9E+09,9E+09,9E+09]];
    PERS robtarget T79:=[[0,0,0],[0.73728,3.31828E-06,0.675588,2.33895E-06],[0,-1,0,0],[9E+09,9E+09,9E+09,9E+09,9E+09,9E+09]];

    PERS robtarget U70:=[[-40.18,-27.37,309.54],[0.507567,-0.694781,-0.175696,-0.478317],[0,1,-2,0],[9E+09,1.24998,21.9999,9E+09,9E+09,9E+09]];
    PERS robtarget U71:=[[-38.65,-23.79,334.77],[0.565972,-0.625405,-0.153135,-0.514874],[0,1,-2,0],[9E+09,1.25001,22,9E+09,9E+09,9E+09]];
    PERS robtarget U72:=[[-84.29,-45.38,314.72],[0.441867,0.0418055,-0.822139,-0.356504],[0,0,-2,0],[9E+09,-24.6237,-70.4231,9E+09,9E+09,9E+09]];
    PERS robtarget U73:=[[-87.46,-79.02,295.66],[0.66022,-0.251573,-0.673606,-0.216976],[-1,0,-2,0],[9E+09,15.9985,-48.8794,9E+09,9E+09,9E+09]];
    PERS robtarget U74:=[[-86.41,-74.16,254.74],[0.653179,-0.269346,-0.66748,-0.235121],[-1,0,-2,0],[9E+09,15.9986,-48.8795,9E+09,9E+09,9E+09]];
    PERS robtarget U75:=[[-87.75,-71.78,236.69],[0.629807,-0.320201,-0.646779,-0.287215],[-1,0,-2,0],[9E+09,15.9985,-48.8795,9E+09,9E+09,9E+09]];
    PERS robtarget U76:=[[-89.49,-33.65,303.7],[0.231731,-0.261825,-0.662764,0.662189],[0,1,-2,0],[9E+09,-10.7,-142.001,9E+09,9E+09,9E+09]];
    PERS robtarget U77:=[[-87.55,-38.98,264.17],[0.231738,-0.261829,-0.662763,0.662186],[0,1,-2,0],[9E+09,-10.7,-132.001,9E+09,9E+09,9E+09]];
    PERS robtarget U78:=[[-84.41,-40.22,244.47],[0.18148,-0.28897,-0.760586,0.552333],[0,1,-2,0],[9E+09,-10.7,-132.001,9E+09,9E+09,9E+09]];
    PERS robtarget U79:=[[0,0,0],[0.73728,3.31828E-06,0.675588,2.33895E-06],[0,-1,0,0],[9E+09,9E+09,9E+09,9E+09,9E+09,9E+09]];

	PERS robtarget SPAG100S:=[[-67.97,-69.57,28.58],[0.707134,1.06993E-06,-5.86054E-07,-0.70708],[0,-1,-1,0],[9E+09,-0.000132496,0.00105351,9E+09,9E+09,9E+09]];
	PERS robtarget SPAG101S:=[[-62.3,56.89,11.57],[0.488131,-0.507412,-0.511746,-0.492319],[-1,0,-2,0],[9E+09,0.00108342,0.000896616,9E+09,9E+09,9E+09]];
	PERS robtarget SPAG102S:=[[191.48,4.49,80.72],[0.00218135,0.703339,-0.710852,2.99839E-05],[0,0,0,0],[9E+09,-7.78641E-06,-4.4762E-05,9E+09,9E+09,9E+09]];
	PERS robtarget SPAG103S:=[[-192.11,4.55,80.36],[0.00203379,0.860454,-0.509526,-0.000190204],[0,1,-1,0],[9E+09,-7.78641E-06,6.55343E-08,9E+09,9E+09,9E+09]];
	PERS robtarget SPAG104S:=[[-381.15,-11.66,205.25],[0.0462075,0.706542,0.0484395,0.7045],[0,0,-2,0],[9E+09,-7.78641E-06,90,9E+09,9E+09,9E+09]];
	PERS robtarget SPAG105S:=[[-326.50,-11.52,205.07],[0.0462054,0.70654,0.0484451,0.704501],[0,0,-2,0],[9E+09,-2.85714E-05,90,9E+09,9E+09,9E+09]];

	PERS robtarget SPAG100E:=[[-67.999,-49.5864,28.5997],[0.793406,-3.31789E-06,5.45271E-06,-0.608694],[-1,-1,-1,0],[9E+09,-0.000132496,0.00105351,9E+09,9E+09,9E+09]];
	PERS robtarget SPAG101E:=[[-81.7987,56.8815,11.5886],[0.488129,-0.507412,-0.511746,-0.49232],[-1,0,-2,0],[9E+09,0.00108342,0.000896616,9E+09,9E+09,9E+09]];
	PERS robtarget SPAG102E:=[[-71.7393,54.6259,-46.492],[0.491476,-0.507002,-0.508426,-0.492853],[-1,0,-2,0],[9E+09,0.00108342,0.000896616,9E+09,9E+09,9E+09]];
	PERS robtarget SPAG103E:=[[-192.11,4.55,80.36],[0.00203379,0.860454,-0.509526,-0.000190204],[0,1,-1,0],[9E+09,-7.78641E-06,6.55343E-08,9E+09,9E+09,9E+09]];
	PERS robtarget SPAG104E:=[[-381.15,-11.66,205.25],[0.0462075,0.706542,0.0484395,0.7045],[0,0,-2,0],[9E+09,-7.78641E-06,90,9E+09,9E+09,9E+09]];
	PERS robtarget SPAG105E:=[[-326.50,-11.52,205.07],[0.0462054,0.70654,0.0484451,0.704501],[0,0,-2,0],[9E+09,-2.85714E-05,90,9E+09,9E+09,9E+09]];

	PERS robtarget SPAH100S:=[[67.97,-69.57,28.58],[0.707134,-7.42093E-07,1.05514E-06,-0.70708],[0,-1,-1,0],[9E+09,-0.000132496,0.00105351,9E+09,9E+09,9E+09]];
	PERS robtarget SPAH101S:=[[62.3,56.89,11.57],[0.488131,-0.507412,-0.511746,-0.492319],[-1,0,-2,0],[9E+09,0.00108342,0.000896616,9E+09,9E+09,9E+09]];
	PERS robtarget SPAH102S:=[[191.48,4.49,80.72],[0.00218135,0.703339,-0.710852,2.99839E-05],[0,0,0,0],[9E+09,-7.78641E-06,-4.4762E-05,9E+09,9E+09,9E+09]];
	PERS robtarget SPAH103S:=[[-192.11,4.55,80.36],[0.00203379,0.860454,-0.509526,-0.000190204],[0,1,-1,0],[9E+09,-7.78641E-06,6.55343E-08,9E+09,9E+09,9E+09]];
	PERS robtarget SPAH104S:=[[-381.15,-11.66,205.25],[0.0462075,0.706542,0.0484395,0.7045],[0,0,-2,0],[9E+09,-7.78641E-06,90,9E+09,9E+09,9E+09]];
	PERS robtarget SPAH105S:=[[-326.50,-11.52,205.07],[0.0462054,0.70654,0.0484451,0.704501],[0,0,-2,0],[9E+09,-2.85714E-05,90,9E+09,9E+09,9E+09]];

	PERS robtarget SPAH100E:=[[67.9709,-49.5835,28.5952],[0.608619,-4.83918E-06,4.64091E-06,-0.793463],[-1,-1,-1,0],[9E+09,-0.000132496,0.00105351,9E+09,9E+09,9E+09]];
	PERS robtarget SPAH101E:=[[81.8033,56.8816,11.5861],[0.48813,-0.507412,-0.511746,-0.49232],[-1,0,-2,0],[9E+09,0.00108342,0.000896616,9E+09,9E+09,9E+09]];
	PERS robtarget SPAH102E:=[[71.7412,54.626,-46.4927],[0.491476,-0.507002,-0.508426,-0.492853],[-1,0,-2,0],[9E+09,0.00108342,0.000896616,9E+09,9E+09,9E+09]];
	PERS robtarget SPAH103E:=[[-192.11,4.55,80.36],[0.00203379,0.860454,-0.509526,-0.000190204],[0,1,-1,0],[9E+09,-7.78641E-06,6.55343E-08,9E+09,9E+09,9E+09]];
	PERS robtarget SPAH104E:=[[-381.15,-11.66,205.25],[0.0462075,0.706542,0.0484395,0.7045],[0,0,-2,0],[9E+09,-7.78641E-06,90,9E+09,9E+09,9E+09]];
	PERS robtarget SPAH105E:=[[-326.50,-11.52,205.07],[0.0462054,0.70654,0.0484451,0.704501],[0,0,-2,0],[9E+09,-2.85714E-05,90,9E+09,9E+09,9E+09]];


	PERS robtarget SPG1S:=[[-141,-50,-195],[0.0111046,-6.45992E-07,2.89574E-06,-0.999939],[0,0,-3,1],[9E+09,0.000231241,90.0014,9E+09,9E+09,9E+09]];
	PERS robtarget SPG2S:=[[-174.15,-106.57,-101.7],[0.559938,0.424139,-0.562162,-0.43652],[-1,0,-3,0],[9E+09,-22.256,-45,9E+09,9E+09,9E+09]];
	PERS robtarget SPG3S:=[[191.48,4.49,80.72],[0.00218135,0.703339,-0.710852,2.99839E-05],[0,0,0,0],[9E+09,-7.78641E-06,-4.4762E-05,9E+09,9E+09,9E+09]];
	PERS robtarget SPG4S:=[[-381.15,-11.66,205.25],[0.0462075,0.706542,0.0484395,0.7045],[0,0,-2,0],[9E+09,-7.78641E-06,90,9E+09,9E+09,9E+09]];
	PERS robtarget SPG5S:=[[-326.50,-11.52,205.07],[0.0462054,0.70654,0.0484451,0.704501],[0,0,-2,0],[9E+09,-2.85714E-05,90,9E+09,9E+09,9E+09]];

	PERS robtarget SPH1S:=[[140.5,-50,-195],[1,-1.47266E-06,9.1079E-07,-0.000163424],[0,1,-2,1],[9E+09,3.49912,-49.2999,9E+09,9E+09,9E+09]];
	PERS robtarget SPH2S:=[[174,-110.9,-95.92],[0.432567,-0.55945,0.432498,-0.559328],[-1,0,-1,0],[9E+09,-22.256,45,9E+09,9E+09,9E+09]];
	PERS robtarget SPH3S:=[[191.48,4.49,80.72],[0.00218135,0.703339,-0.710852,2.99839E-05],[0,0,0,0],[9E+09,-7.78641E-06,-4.4762E-05,9E+09,9E+09,9E+09]];
	PERS robtarget SPH4S:=[[-381.15,-11.66,205.25],[0.0462075,0.706542,0.0484395,0.7045],[0,0,-2,0],[9E+09,-7.78641E-06,90,9E+09,9E+09,9E+09]];
	PERS robtarget SPH5S:=[[-326.50,-11.52,205.07],[0.0462054,0.70654,0.0484451,0.704501],[0,0,-2,0],[9E+09,-2.85714E-05,90,9E+09,9E+09,9E+09]];

	PERS robtarget SPG40S:=[[-30.01,40.74,-178.27],[0.500201,-0.49991,0.499802,-0.500087],[-1,0,-1,0],[9E+09,-21,49,9E+09,9E+09,9E+09]];
	PERS robtarget SPG41S:=[[-146.89,-9.40,-247.89],[0.51934,-0.422004,0.568784,-0.47821],[-1,1,-2,0],[9E+09,-7.78641E-06,89.9702,9E+09,9E+09,9E+09]];
	PERS robtarget SPG42S:=[[-145.55,-9.97,-180.38],[0.519156,-0.421915,0.568942,-0.4783],[-1,1,-2,0],[9E+09,-2.85714E-05,89.9997,9E+09,9E+09,9E+09]];
	PERS robtarget SPG43S:=[[-103.2,43.24,20],[0.0301262,-0.0301245,0.706453,0.706477],[-1,1,-4,0],[9E+09,4.13336,88.0983,9E+09,9E+09,9E+09]];
	PERS robtarget SPG44S:=[[-188.40,-8.41,-78.39],[0.154298,0.039851,-0.0944107,-0.982696],[-1,2,-4,0],[9E+09,4.2588,88.0441,9E+09,9E+09,9E+09]];
	PERS robtarget SPG45S:=[[-145.38,-10.22,-212.32],[0.519143,-0.421909,0.568953,-0.478308],[-1,1,-2,0],[9E+09,2.3391E-05,89.9997,9E+09,9E+09,9E+09]];
	PERS robtarget SPG46S:=[[-146.52,-10.10,-258.78],[0.519155,-0.421914,0.568944,-0.478301],[-1,1,-2,0],[9E+09,3.99997,90.0007,9E+09,9E+09,9E+09]];
	PERS robtarget SPG47S:=[[-137.66,-5.81,-273.33],[0.555796,-0.502552,0.280066,-0.600081],[-1,1,-3,0],[9E+09,4.99963,89.9996,9E+09,9E+09,9E+09]];
	PERS robtarget SPG48S:=[[-139.61,-6.45,-267.37],[0.614745,-0.423292,0.202072,-0.634098],[-1,1,-3,0],[9E+09,4.99967,89.9996,9E+09,9E+09,9E+09]];
    PERS robtarget SPG49S:=[[-137.11,-12.14,-266.42],[0.588376,-0.357559,0.267329,-0.674168],[-1,1,-3,0],[9E+09,4.99963,89.9996,9E+09,9E+09,9E+09]];

	PERS robtarget SPG50S:=[[-107.912,-55.0006,-174.42],[0.429907,-0.561601,0.429761,-0.561329],[-1,-4,2,0],[9E+09,-4.93563E-05,90.0001,9E+09,9E+09,9E+09]];
	PERS robtarget SPG51S:=[[-30.04,-116.92,-104.27],[0.426573,-0.563924,0.426615,-0.563937],[-1,-4,2,0],[9E+09,0,90,9E+09,9E+09,9E+09]];
	PERS robtarget SPG52S:=[[-111.69,-34.90,-191.63],[0.199681,0.600584,-0.383339,-0.672666],[-1,-1,-3,0],[9E+09,1.99996,-80.9999,9E+09,9E+09,9E+09]];
	PERS robtarget SPG53S:=[[-107.46,-12.68,-198.90],[0.147052,0.541523,-0.416523,-0.715289],[-1,-1,-3,0],[9E+09,1.99998,-80.9998,9E+09,9E+09,9E+09]];
	PERS robtarget SPG54S:=[[-112.36,-85.11,-182.80],[0.227553,0.58966,-0.343343,-0.694721],[-1,-1,-3,0],[9E+09,3.60003,-90,9E+09,9E+09,9E+09]];
	PERS robtarget SPG55S:=[[-107.912,-55.0007,-176.23],[0.429906,-0.561601,0.429761,-0.561329],[-1,-4,2,0],[9E+09,-4.93563E-05,90.0001,9E+09,9E+09,9E+09]];
	PERS robtarget SPG56S:=[[-122.912,-55.0006,-197.106],[0.432907,-0.558815,0.432727,-0.559522],[-1,-4,2,0],[9E+09,-7.78641E-06,89.9999,9E+09,9E+09,9E+09]];
	PERS robtarget SPG57S:=[[-112.34,-84.95,-182.13],[0.227565,0.589671,-0.343343,-0.694709],[-1,-1,-3,0],[9E+09,-2.49997,-85,9E+09,9E+09,9E+09]];
	PERS robtarget SPG58S:=[[-109.81,-49.62,-189.01],[0.227566,0.589661,-0.343352,-0.694712],[-1,-1,-3,0],[9E+09,-2.49995,-85,9E+09,9E+09,9E+09]];
    PERS robtarget SPG59S:=[[-107.56,-12.61,-197.57],[0.086332,0.57466,-0.369462,-0.725129],[-1,-1,-3,0],[9E+09,2.00033,-81,9E+09,9E+09,9E+09]];

	PERS robtarget SPH40S:=[[16.41,38.74,-176.58],[0.167188,-0.687057,-0.167188,0.687058],[-1,2,-2,0],[9E+09,-21,-49,9E+09,9E+09,9E+09]];
	PERS robtarget SPH41S:=[[146.94,-7.14,-246.98],[0.639919,-0.321982,-0.598348,0.358905],[-1,1,-2,0],[9E+09,0.000594977,-90.0001,9E+09,9E+09,9E+09]];
	PERS robtarget SPH42S:=[[147.91,-8.00,-179.17],[0.639921,-0.321992,-0.598341,0.358904],[-1,1,-2,0],[9E+09,2.3391E-05,-90,9E+09,9E+09,9E+09]];
	PERS robtarget SPH43S:=[[101.69,47.25,20],[0.711934,-0.702073,-0.0109009,-0.011159],[-1,2,-2,1],[9E+09,9.61384E-05,-90.0002,9E+09,9E+09,9E+09]];
	PERS robtarget SPH44S:=[[195.40,-15.09,-77.59],[0.998541,-0.0321173,0.0380987,0.0208426],[-1,1,-3,1],[9E+09,9.61384E-05,-90.0002,9E+09,9E+09,9E+09]];
	PERS robtarget SPH45S:=[[146.47,-4.42,-217.18],[0.639919,-0.321987,-0.598345,0.358905],[-1,1,-2,0],[9E+09,-7.78641E-06,-90.0001,9E+09,9E+09,9E+09]];
	PERS robtarget SPH46S:=[[145.71,-4.23,-254.81],[0.639921,-0.322004,-0.598339,0.358897],[-1,1,-2,0],[9E+09,-0.000496233,-89.9999,9E+09,9E+09,9E+09]];
	PERS robtarget SPH47S:=[[139.68,-17.98,-269.29],[0.710161,-0.341994,-0.385916,0.479356],[0,2,-3,0],[9E+09,2.3391E-05,-90.0001,9E+09,9E+09,9E+09]];
	PERS robtarget SPH48S:=[[138.28,-10.67,-270.41],[0.766529,-0.431199,-0.233929,0.414463],[0,3,-4,0],[9E+09,-7.78641E-06,-90,9E+09,9E+09,9E+09]];
    PERS robtarget SPH49S:=[[139.13,-10.80,-275.62],[0.650536,-0.590981,-0.312159,0.360698],[-1,3,-4,0],[9E+09,2.3391E-05,-90.0001,9E+09,9E+09,9E+09]];

	PERS robtarget SPH50S:=[[107.512,-50.4998,-175.53],[0.433111,-0.559144,-0.432622,0.559117],[-1,-2,1,0],[9E+09,-7.78641E-06,-90.0014,9E+09,9E+09,9E+09]];
	PERS robtarget SPH51S:=[[29.81,-104.93,-89.01],[0.430451,-0.560649,-0.430882,0.561004],[-1,-2,1,0],[9E+09,-7.78641E-06,-90,9E+09,9E+09,9E+09]];
	PERS robtarget SPH52S:=[[112.29,-35.29,-195.82],[0.569733,-0.551396,0.486259,-0.367317],[-1,1,-2,0],[9E+09,-1.99998,90,9E+09,9E+09,9E+09]];
	PERS robtarget SPH53S:=[[112.73,-14.85,-200.79],[0.655493,-0.523213,0.402555,-0.36678],[-1,1,-3,0],[9E+09,-2.00001,90,9E+09,9E+09,9E+09]];
	PERS robtarget SPH54S:=[[114.46,-84.77,-184.60],[0.56263,-0.501185,0.518999,-0.403612],[-1,1,-2,0],[9E+09,-2.50652,89.9999,9E+09,9E+09,9E+09]];
	PERS robtarget SPH55S:=[[107.512,-50.4998,-176.38],[0.433112,-0.559141,-0.432624,0.559117],[-1,-2,1,0],[9E+09,-7.78641E-06,-90.0014,9E+09,9E+09,9E+09]];
	PERS robtarget SPH56S:=[[122.512,-50.4998,-199.777],[0.431778,-0.560174,-0.433953,0.558085],[-1,-2,1,0],[9E+09,-7.78641E-06,-90.0014,9E+09,9E+09,9E+09]];
	PERS robtarget SPH57S:=[[115.69,-85.08,-184.48],[0.56287,-0.500912,0.518809,-0.40386],[-1,1,-2,0],[9E+09,-2.5065,83.6248,9E+09,9E+09,9E+09]];
	PERS robtarget SPH58S:=[[112.49,-47.87,-191.60],[0.582601,-0.505669,0.492895,-0.402407],[-1,1,-2,0],[9E+09,-2.5,83.6249,9E+09,9E+09,9E+09]];
    PERS robtarget SPH59S:=[[113.16,-16.51,-199.66],[0.6797,-0.497081,0.382243,-0.380539],[-1,1,-3,0],[9E+09,-2.00058,89.9997,9E+09,9E+09,9E+09]];

	PERS robtarget SPJ1S:=[[3.49,-27.31,-239.82],[0.501774,-0.501858,0.498241,0.498115],[-1,0,-4,0],[9E+09,18.5,0.000336272,9E+09,9E+09,9E+09]];
	PERS robtarget SPJ2S:=[[7.35,-49.05,-116.41],[0.724945,-0.0658516,-0.0586655,-0.683138],[-1,0,-2,0],[9E+09,20.1,0.000448341,9E+09,9E+09,9E+09]];
	PERS robtarget SPJ3S:=[[191.48,4.49,80.72],[0.00218135,0.703339,-0.710852,2.99839E-05],[0,0,0,0],[9E+09,-7.78641E-06,-4.4762E-05,9E+09,9E+09,9E+09]];
	PERS robtarget SPJ4S:=[[-326.50,-11.52,205.07],[0.0462054,0.70654,0.0484451,0.704501],[0,0,-2,0],[9E+09,-2.85714E-05,90,9E+09,9E+09,9E+09]];
	PERS robtarget SPJ5S:=[[0,0,0],[0.73728,3.31828E-06,0.675588,2.33895E-06],[0,-1,0,0],[9E+09,9E+09,9E+09,9E+09,9E+09,9E+09]];

	PERS robtarget SPK1S:=[[192.08,-8.78,283.74],[0.0021613,0.781238,-0.624231,-1.93188E-05],[0,1,-1,0],[9E+09,-20,-20,9E+09,9E+09,9E+09]];
	PERS robtarget SPK2S:=[[-192.69,-8.97,283.97],[0.00211019,0.781244,-0.624224,3.11178E-05],[0,0,0,0],[9E+09,-20,-20,9E+09,9E+09,9E+09]];
	PERS robtarget SPK3S:=[[191.48,4.49,80.72],[0.00218135,0.703339,-0.710852,2.99839E-05],[0,0,0,0],[9E+09,-7.78641E-06,-4.4762E-05,9E+09,9E+09,9E+09]];
	PERS robtarget SPK4S:=[[-326.50,-11.52,205.07],[0.0462054,0.70654,0.0484451,0.704501],[0,0,-2,0],[9E+09,-2.85714E-05,90,9E+09,9E+09,9E+09]];
	PERS robtarget SPK5S:=[[0,0,0],[0.73728,3.31828E-06,0.675588,2.33895E-06],[0,-1,0,0],[9E+09,9E+09,9E+09,9E+09,9E+09,9E+09]];


    PERS robtarget SPP1S:=[[54.43,-22.61,217.23],[0.497307,0.497307,-0.502678,0.502678],[-1,2,-4,1],[9E+09,-18.5,180,9E+09,9E+09,9E+09]];
    PERS robtarget SPP2S:=[[-14.69,15.26,189.65],[0.500211,-0.499818,-0.500175,0.499796],[0,2,-2,1],[9E+09,-18,180,9E+09,9E+09,9E+09]];
    PERS robtarget SPP3S:=[[159.54,-76.01,226.65],[0.497306,0.497308,-0.502678,0.502679],[-1,2,-4,1],[9E+09,-26,180,9E+09,9E+09,9E+09]];
    PERS robtarget SPP4S:=[[0,0,0],[0.73728,3.31828E-06,0.675588,2.33895E-06],[0,-1,0,0],[9E+09,9E+09,9E+09,9E+09,9E+09,9E+09]];


    PERS robtarget SPR1S:=[[1.9,-5.85,-219.73],[0.000407167,0.000422533,0.719285,-0.694715],[-1,1,-2,0],[9E+09,24.5,180,9E+09,9E+09,9E+09]];
    PERS robtarget SPR2S:=[[-159.44,-74.83,-181.34],[3.01668E-05,3.19296E-05,0.707148,-0.707066],[-1,1,-3,0],[9E+09,21.7,180,9E+09,9E+09,9E+09]];
    PERS robtarget SPR5S:=[[102.86,33.37,-183.4],[0.524726,0.47387,0.524811,0.474008],[-1,1,-5,0],[9E+09,21.7,180,9E+09,9E+09,9E+09]];

    PERS robtarget SPT11S:=[[19.7,-60.19,144.53],[0.645229,-0.547175,-0.345611,-0.405997],[0,1,-2,0],[9E+09,31,0.00177075,9E+09,9E+09,9E+09]];
    PERS robtarget SPT12S:=[[-136.88,-59.09,181.65],[0.676751,-0.538459,-0.312595,-0.39288],[-1,0,-2,0],[9E+09,34,0,9E+09,9E+09,9E+09]];
    PERS robtarget SPT20S:=[[36.16,-64.39,246.22],[0.761026,-0.577575,-0.178341,-0.235461],[0,2,-4,0],[9E+09,-13.4,0.000336272,9E+09,9E+09,9E+09]];


    PERS robtarget SPT40S:=[[107.57,-53.14,246.21],[0.563521,-0.427494,-0.563007,0.427454],[0,1,-2,0],[9E+09,1.13372,-89.2773,9E+09,9E+09,9E+09]];
    PERS robtarget SPT41S:=[[141.58,-28.44,129.33],[0.513522,-0.525442,-0.475383,0.483962],[0,1,-2,0],[9E+09,1.13303,-89.2777,9E+09,9E+09,9E+09]];
    PERS robtarget SPT42S:=[[141.70,-20.86,130.12],[0.513529,-0.525447,-0.475377,0.483954],[0,1,-2,0],[9E+09,1.13303,-89.2777,9E+09,9E+09,9E+09]];
    PERS robtarget SPT43S:=[[138.20,-32.60,129.04],[0.513543,-0.525446,-0.475376,0.483941],[0,1,-2,0],[9E+09,1.13305,-89.2778,9E+09,9E+09,9E+09]];
	PERS robtarget SPT44S:=[[139.51,-27.86,128.84],[0.513549,-0.525446,-0.475376,0.483936],[0,1,-2,0],[9E+09,1.13306,-89.2777,9E+09,9E+09,9E+09]];

    PERS robtarget SPT50S:=[[-107.80,-53.92,245.24],[0.565308,-0.424678,0.56535,-0.4248],[0,2,-3,0],[9E+09,1.01673,89.559,9E+09,9E+09,9E+09]];
    PERS robtarget SPT51S:=[[-134.41,-21.31,130.00],[0.271508,-0.629436,0.285253,-0.66987],[0,1,-2,0],[9E+09,1.01926,89.5582,9E+09,9E+09,9E+09]];
    PERS robtarget SPT52S:=[[-134.26,-30.69,129.15],[0.271506,-0.629435,0.28525,-0.669874],[0,1,-2,0],[9E+09,1.01926,89.5581,9E+09,9E+09,9E+09]];
    PERS robtarget SPT53S:=[[-137.13,-21.49,129.92],[0.2715,-0.629431,0.285247,-0.669881],[0,1,-2,0],[9E+09,1.01926,89.5581,9E+09,9E+09,9E+09]];
    PERS robtarget SPT54S:=[[-137.13,-21.49,129.92],[0.2715,-0.629431,0.285247,-0.669881],[0,1,-2,0],[9E+09,1.01926,89.5581,9E+09,9E+09,9E+09]];



	PERS robtarget SPG1E:=[[-120.5,-50,-195],[0.0111046,-6.45992E-07,2.89574E-06,-0.999939],[0,0,-3,1],[9E+09,0.000231241,90.0014,9E+09,9E+09,9E+09]];
	PERS robtarget SPG2E:=[[-173.83,-82.6502,-108.12],[0.559938,0.424139,-0.562162,-0.43652],[-1,0,-3,0],[9E+09,-22.256,-45,9E+09,9E+09,9E+09]];
	PERS robtarget SPG3E:=[[191.48,4.49,80.72],[0.00218135,0.703339,-0.710852,2.99839E-05],[0,0,0,0],[9E+09,-7.78641E-06,-4.4762E-05,9E+09,9E+09,9E+09]];
	PERS robtarget SPG4E:=[[-381.15,-11.66,205.25],[0.0462075,0.706542,0.0484395,0.7045],[0,0,-2,0],[9E+09,-7.78641E-06,90,9E+09,9E+09,9E+09]];
	PERS robtarget SPG5E:=[[-326.50,-11.52,205.07],[0.0462054,0.70654,0.0484451,0.704501],[0,0,-2,0],[9E+09,-2.85714E-05,90,9E+09,9E+09,9E+09]];

	PERS robtarget SPH1E:=[[120.50,-50.00,-195.00],[1,-1.47266E-06,9.1079E-07,-0.000163424],[0,1,-2,1],[9E+09,3.49912,-49.2999,9E+09,9E+09,9E+09]];
	PERS robtarget SPH2E:=[[173.99,-82.2303,-103.37],[0.432567,-0.559449,0.432498,-0.559328],[-1,0,-1,0],[9E+09,-22.256,45,9E+09,9E+09,9E+09]];
	PERS robtarget SPH3E:=[[191.48,4.49,80.72],[0.00218135,0.703339,-0.710852,2.99839E-05],[0,0,0,0],[9E+09,-7.78641E-06,-4.4762E-05,9E+09,9E+09,9E+09]];
	PERS robtarget SPH4E:=[[-381.15,-11.66,205.25],[0.0462075,0.706542,0.0484395,0.7045],[0,0,-2,0],[9E+09,-7.78641E-06,90,9E+09,9E+09,9E+09]];
	PERS robtarget SPH5E:=[[-326.50,-11.52,205.07],[0.0462054,0.70654,0.0484451,0.704501],[0,0,-2,0],[9E+09,-2.85714E-05,90,9E+09,9E+09,9E+09]];

	PERS robtarget SPG40E:=[[-30,9.84991,-178.27],[0.500201,-0.49991,0.499802,-0.500087],[-1,-1,-1,0],[9E+09,-21,49,9E+09,9E+09,9E+09]];
	PERS robtarget SPG41E:=[[-146.89,-9.40,-247.89],[0.51934,-0.422004,0.568784,-0.47821],[-1,1,-2,0],[9E+09,-7.78641E-06,89.9702,9E+09,9E+09,9E+09]];
	PERS robtarget SPG42E:=[[-145.55,-9.97,-180.38],[0.519156,-0.421915,0.568942,-0.4783],[-1,1,-2,0],[9E+09,-2.85714E-05,89.9997,9E+09,9E+09,9E+09]];
	PERS robtarget SPG43E:=[[-102.27,47.80,-1.54],[0.707106,-0.707107,-0.000325448,-0.000324941],[-1,0,-1,0],[9E+09,-22.256,-46.3804,9E+09,9E+09,9E+09]];
	PERS robtarget SPG44E:=[[-164.40,-8.37,-78.24],[0.154283,0.0398477,-0.0944108,-0.982699],[-1,2,-4,0],[9E+09,4.2581,88.0442,9E+09,9E+09,9E+09]];
	PERS robtarget SPG45E:=[[-145.38,-10.22,-212.32],[0.519143,-0.421909,0.568953,-0.478308],[-1,1,-2,0],[9E+09,2.3391E-05,89.9997,9E+09,9E+09,9E+09]];
	PERS robtarget SPG46E:=[[-146.52,-10.10,-258.78],[0.519155,-0.421914,0.568944,-0.478301],[-1,1,-2,0],[9E+09,3.99997,90.0007,9E+09,9E+09,9E+09]];
	PERS robtarget SPG47E:=[[-137.66,-5.81,-273.33],[0.555796,-0.502552,0.280066,-0.600081],[-1,1,-3,0],[9E+09,4.99963,89.9996,9E+09,9E+09,9E+09]];
	PERS robtarget SPG48E:=[[-139.61,-6.45,-267.37],[0.614745,-0.423292,0.202072,-0.634098],[-1,1,-3,0],[9E+09,4.99967,89.9996,9E+09,9E+09,9E+09]];
    PERS robtarget SPG49E:=[[-137.11,-12.14,-266.42],[0.588376,-0.357559,0.267329,-0.674168],[-1,1,-3,0],[9E+09,4.99963,89.9996,9E+09,9E+09,9E+09]];

	PERS robtarget SPG50E:=[[-107.912,-55.0006,-154.42],[0.429907,-0.561601,0.429761,-0.561329],[-1,-4,2,0],[9E+09,-4.93563E-05,90.0001,9E+09,9E+09,9E+09]];
	PERS robtarget SPG51E:=[[-30.0399,-85.0005,-113.3],[0.426574,-0.563924,0.426615,-0.563937],[-1,-4,2,0],[9E+09,0,90,9E+09,9E+09,9E+09]];
	PERS robtarget SPG52E:=[[-111.69,-34.90,-191.63],[0.199681,0.600584,-0.383339,-0.672666],[-1,-1,-3,0],[9E+09,1.99996,-80.9999,9E+09,9E+09,9E+09]];
	PERS robtarget SPG53E:=[[-107.46,-12.68,-198.90],[0.147052,0.541523,-0.416523,-0.715289],[-1,-1,-3,0],[9E+09,1.99998,-80.9998,9E+09,9E+09,9E+09]];
	PERS robtarget SPG54E:=[[-112.36,-85.11,-182.80],[0.227553,0.58966,-0.343343,-0.694721],[-1,-1,-3,0],[9E+09,3.60003,-90,9E+09,9E+09,9E+09]];
	PERS robtarget SPG55E:=[[-107.912,-55.0007,-151.23],[0.429906,-0.561601,0.429761,-0.561329],[-1,-4,2,0],[9E+09,-4.93563E-05,90.0001,9E+09,9E+09,9E+09]];
	PERS robtarget SPG56E:=[[-107.912,-55.0006,-197.106],[0.432907,-0.558815,0.432727,-0.559522],[-1,-4,2,0],[9E+09,-7.78641E-06,89.9999,9E+09,9E+09,9E+09]];
	PERS robtarget SPG57E:=[[-112.34,-84.95,-182.13],[0.227565,0.589671,-0.343343,-0.694709],[-1,-1,-3,0],[9E+09,-2.49997,-85,9E+09,9E+09,9E+09]];
	PERS robtarget SPG58E:=[[-109.81,-49.62,-189.01],[0.227566,0.589661,-0.343352,-0.694712],[-1,-1,-3,0],[9E+09,-2.49995,-85,9E+09,9E+09,9E+09]];
    PERS robtarget SPG59E:=[[-107.56,-12.61,-197.57],[0.086332,0.57466,-0.369462,-0.725129],[-1,-1,-3,0],[9E+09,2.00033,-81,9E+09,9E+09,9E+09]];




	PERS robtarget SPH40E:=[[16.4101,9.50021,-179.23],[0.167189,-0.687057,-0.167188,0.687058],[-1,2,-2,0],[9E+09,-21,-49,9E+09,9E+09,9E+09]];
	PERS robtarget SPH41E:=[[146.94,-7.14,-246.98],[0.639919,-0.321982,-0.598348,0.358905],[-1,1,-2,0],[9E+09,0.000594977,-90.0001,9E+09,9E+09,9E+09]];
	PERS robtarget SPH42E:=[[147.91,-8.00,-179.17],[0.639921,-0.321992,-0.598341,0.358904],[-1,1,-2,0],[9E+09,2.3391E-05,-90,9E+09,9E+09,9E+09]];
	PERS robtarget SPH43E:=[[102,41.3997,-1.41008],[0.666755,-0.666753,0.235454,0.235454],[-1,1,-2,0],[9E+09,-22.256,45,9E+09,9E+09,9E+09]];
	PERS robtarget SPH44E:=[[168.27,-15.28,-77.70],[0.99854,-0.0321044,0.0381283,0.0208737],[-1,1,-3,1],[9E+09,0.000615762,-90,9E+09,9E+09,9E+09]];
	PERS robtarget SPH45E:=[[146.47,-4.42,-217.18],[0.639919,-0.321987,-0.598345,0.358905],[-1,1,-2,0],[9E+09,-7.78641E-06,-90.0001,9E+09,9E+09,9E+09]];
	PERS robtarget SPH46E:=[[145.71,-4.23,-254.81],[0.639921,-0.322004,-0.598339,0.358897],[-1,1,-2,0],[9E+09,-0.000496233,-89.9999,9E+09,9E+09,9E+09]];
	PERS robtarget SPH47E:=[[139.68,-17.98,-269.29],[0.710161,-0.341994,-0.385916,0.479356],[0,2,-3,0],[9E+09,2.3391E-05,-90.0001,9E+09,9E+09,9E+09]];
	PERS robtarget SPH48E:=[[138.28,-10.67,-270.41],[0.766529,-0.431199,-0.233929,0.414463],[0,3,-4,0],[9E+09,-7.78641E-06,-90,9E+09,9E+09,9E+09]];
    PERS robtarget SPH49E:=[[139.13,-10.80,-275.62],[0.650536,-0.590981,-0.312159,0.360698],[-1,3,-4,0],[9E+09,2.3391E-05,-90.0001,9E+09,9E+09,9E+09]];

	PERS robtarget SPH50E:=[[107.512,-50.4998,-155.53],[0.433111,-0.559144,-0.432622,0.559117],[-1,-2,1,0],[9E+09,-7.78641E-06,-90.0014,9E+09,9E+09,9E+09]];
	PERS robtarget SPH51E:=[[29.7898,-80.4998,-95.5398],[0.430451,-0.560649,-0.430882,0.561004],[-1,-2,1,0],[9E+09,-7.78641E-06,-90,9E+09,9E+09,9E+09]];
	PERS robtarget SPH52E:=[[112.29,-35.29,-195.82],[0.569733,-0.551396,0.486259,-0.367317],[-1,1,-2,0],[9E+09,-1.99998,90,9E+09,9E+09,9E+09]];
	PERS robtarget SPH53E:=[[112.73,-14.85,-200.79],[0.655493,-0.523213,0.402555,-0.36678],[-1,1,-3,0],[9E+09,-2.00001,90,9E+09,9E+09,9E+09]];
	PERS robtarget SPH54E:=[[114.46,-84.77,-184.60],[0.56263,-0.501185,0.518999,-0.403612],[-1,1,-2,0],[9E+09,-2.50652,89.9999,9E+09,9E+09,9E+09]];
	PERS robtarget SPH55E:=[[107.512,-50.4998,-151.38],[0.433112,-0.559141,-0.432624,0.559117],[-1,-2,1,0],[9E+09,-7.78641E-06,-90.0014,9E+09,9E+09,9E+09]];
	PERS robtarget SPH56E:=[[107.512,-50.4998,-199.777],[0.431778,-0.560174,-0.433953,0.558085],[-1,-2,1,0],[9E+09,-7.78641E-06,-90.0014,9E+09,9E+09,9E+09]];
	PERS robtarget SPH57E:=[[115.69,-85.08,-184.48],[0.56287,-0.500912,0.518809,-0.40386],[-1,1,-2,0],[9E+09,-2.5065,83.6248,9E+09,9E+09,9E+09]];
	PERS robtarget SPH58E:=[[112.49,-47.87,-191.60],[0.582601,-0.505669,0.492895,-0.402407],[-1,1,-2,0],[9E+09,-2.5,83.6249,9E+09,9E+09,9E+09]];
    PERS robtarget SPH59E:=[[113.16,-16.51,-199.66],[0.6797,-0.497081,0.382243,-0.380539],[-1,1,-3,0],[9E+09,-2.00058,89.9997,9E+09,9E+09,9E+09]];

	PERS robtarget SPJ1E:=[[3.43,-21.6002,-231.46],[0.501776,-0.501857,0.498241,0.498113],[-1,-1,-4,0],[9E+09,20.3,0,9E+09,9E+09,9E+09]];
	PERS robtarget SPJ2E:=[[6.82014,-19.8099,-132.9],[0.700928,-0.0937349,-0.0941318,-0.700752],[-1,0,-2,0],[9E+09,20.3,0.000448341,9E+09,9E+09,9E+09]];
	PERS robtarget SPJ3E:=[[81.08,-36.56,-245.78],[0.631686,-0.318702,-0.318403,-0.63089],[-1,0,-2,0],[9E+09,20.3,-0.000762002,9E+09,9E+09,9E+09]];
	PERS robtarget SPJ4E:=[[-326.50,-11.52,205.07],[0.0462054,0.70654,0.0484451,0.704501],[0,0,-2,0],[9E+09,-2.85714E-05,90,9E+09,9E+09,9E+09]];
	PERS robtarget SPJ5E:=[[0,0,0],[0.73728,3.31828E-06,0.675588,2.33895E-06],[0,-1,0,0],[9E+09,9E+09,9E+09,9E+09,9E+09,9E+09]];

	PERS robtarget SPK1E:=[[192.08,-8.78,283.74],[0.0021613,0.781238,-0.624231,-1.93188E-05],[0,1,-1,0],[9E+09,-20,-20,9E+09,9E+09,9E+09]];
	PERS robtarget SPK2E:=[[-192.69,-8.97,283.97],[0.00211019,0.781244,-0.624224,3.11178E-05],[0,0,0,0],[9E+09,-20,-20,9E+09,9E+09,9E+09]];
	PERS robtarget SPK3E:=[[191.48,4.49,80.72],[0.00218135,0.703339,-0.710852,2.99839E-05],[0,0,0,0],[9E+09,-7.78641E-06,-4.4762E-05,9E+09,9E+09,9E+09]];
	PERS robtarget SPK4E:=[[-326.50,-11.52,205.07],[0.0462054,0.70654,0.0484451,0.704501],[0,0,-2,0],[9E+09,-2.85714E-05,90,9E+09,9E+09,9E+09]];
	PERS robtarget SPK5E:=[[0,0,0],[0.73728,3.31828E-06,0.675588,2.33895E-06],[0,-1,0,0],[9E+09,9E+09,9E+09,9E+09,9E+09,9E+09]];

    PERS robtarget SPP1E:=[[54.6482,-22.61,206.256],[0.648623,0.648676,-0.281504,0.281537],[0,2,-4,1],[9E+09,-18.5,180,9E+09,9E+09,9E+09]];
    PERS robtarget SPP2E:=[[-14.7301,-8.96205,189.842],[0.609967,-0.357674,-0.610096,0.357482],[0,2,-3,1],[9E+09,-18.5,180,9E+09,9E+09,9E+09]];
    PERS robtarget SPP1EE:=[[0,0,0],[0.73728,3.31828E-06,0.675588,2.33895E-06],[0,-1,0,0],[9E+09,9E+09,9E+09,9E+09,9E+09,9E+09]];
    PERS robtarget SPP2EE:=[[0,0,0],[0.73728,3.31828E-06,0.675588,2.33895E-06],[0,-1,0,0],[9E+09,9E+09,9E+09,9E+09,9E+09,9E+09]];
    PERS robtarget SPP3E:=[[128.557,-75.9842,226.367],[0.613535,0.613623,-0.351465,0.351446],[-1,2,-4,1],[9E+09,-18.5,180,9E+09,9E+09,9E+09]];
    PERS robtarget SPP4E:=[[0,0,0],[0.73728,3.31828E-06,0.675588,2.33895E-06],[0,-1,0,0],[9E+09,9E+09,9E+09,9E+09,9E+09,9E+09]];

    PERS robtarget SPR1E:=[[1.88012,-5.85,-205.02],[0.000408208,0.000422279,0.719285,-0.694715],[-1,1,-2,0],[9E+09,24.5,180,9E+09,9E+09,9E+09]];
    PERS robtarget SPR2E:=[[-129.443,-74.8259,-181.341],[3.04174E-05,3.18299E-05,0.707148,-0.707066],[-1,1,-2,0],[9E+09,24.5,180,9E+09,9E+09,9E+09]];
    PERS robtarget SPR5E:=[[64.8922,28.1375,-130.353],[0.524759,0.473887,0.524775,0.473994],[-1,1,-5,0],[9E+09,24,180,9E+09,9E+09,9E+09]];

    PERS robtarget SPR10S:=[[1.9,-5.85,-219.73],[0.000407001,0.000422495,0.719285,-0.694715],[-1,1,-2,0],[9E+09,24.5,180,9E+09,9E+09,9E+09]];
    PERS robtarget SPR10E:=[[1.90004,-5.85,-206.73],[0.000408267,0.000422671,0.719285,-0.694715],[-1,1,-2,0],[9E+09,24.5,180,9E+09,9E+09,9E+09]];


    PERS robtarget SPT11E:=[[19.75,-62.1,156.16],[0.645232,-0.547177,-0.345607,-0.405992],[0,1,-2,0],[9E+09,31,0.00177075,9E+09,9E+09,9E+09]];
    PERS robtarget SPT12E:=[[-116.834,-59.0559,181.294],[0.676623,-0.538582,-0.31265,-0.392887],[-1,0,-2,0],[9E+09,34,0.000130474,9E+09,9E+09,9E+09]];
    PERS robtarget SPT20E:=[[35.87,-61.22,235.23],[0.761025,-0.577576,-0.178341,-0.235459],[0,2,-4,0],[9E+09,-13.4,0.000489094,9E+09,9E+09,9E+09]];
    PERS robtarget SPT21E:=[[0,0,0],[0.73728,3.31828E-06,0.675588,2.33895E-06],[0,-1,0,0],[9E+09,9E+09,9E+09,9E+09,9E+09,9E+09]];
    PERS robtarget SPT22E:=[[0,0,0],[0.73728,3.31828E-06,0.675588,2.33895E-06],[0,-1,0,0],[9E+09,9E+09,9E+09,9E+09,9E+09,9E+09]];
    PERS robtarget SPT55S:=[[59.3,-67.48,175.82],[0.553373,-0.440299,-0.440226,-0.553279],[-1,0,-2,0],[9E+09,34,0,9E+09,9E+09,9E+09]];
    PERS robtarget SPT55E:=[[59.8728,-67.48,162.245],[0.553259,-0.440584,-0.440109,-0.553258],[-1,0,-2,0],[9E+09,34,-0.000116078,9E+09,9E+09,9E+09]];



    PERS robtarget SPT40E:=[[107.57,-50.0555,236.72],[0.5634,-0.427668,-0.562934,0.427534],[0,1,-2,0],[9E+09,1.13373,-89.2771,9E+09,9E+09,9E+09]];
    PERS robtarget SPT41E:=[[141.58,-28.44,129.33],[0.513522,-0.525442,-0.475383,0.483962],[0,1,-2,0],[9E+09,1.13303,-89.2777,9E+09,9E+09,9E+09]];
    PERS robtarget SPT42E:=[[141.70,-20.86,130.12],[0.513529,-0.525447,-0.475377,0.483954],[0,1,-2,0],[9E+09,1.13303,-89.2777,9E+09,9E+09,9E+09]];
    PERS robtarget SPT43E:=[[138.20,-32.60,129.04],[0.513543,-0.525446,-0.475376,0.483941],[0,1,-2,0],[9E+09,1.13305,-89.2778,9E+09,9E+09,9E+09]];
	PERS robtarget SPT44E:=[[139.51,-27.86,128.84],[0.513549,-0.525446,-0.475376,0.483936],[0,1,-2,0],[9E+09,1.13306,-89.2777,9E+09,9E+09,9E+09]];

    PERS robtarget SPT50E:=[[-107.8,-51.1919,236.57],[0.565234,-0.424692,0.565261,-0.425003],[0,2,-3,0],[9E+09,1.01672,89.559,9E+09,9E+09,9E+09]];
    PERS robtarget SPT51E:=[[-134.41,-21.31,130.00],[0.271508,-0.629436,0.285253,-0.66987],[0,1,-2,0],[9E+09,1.01926,89.5582,9E+09,9E+09,9E+09]];
    PERS robtarget SPT52E:=[[-134.26,-30.69,129.15],[0.271506,-0.629435,0.28525,-0.669874],[0,1,-2,0],[9E+09,1.01926,89.5581,9E+09,9E+09,9E+09]];
    PERS robtarget SPT53E:=[[-137.13,-21.49,129.92],[0.2715,-0.629431,0.285247,-0.669881],[0,1,-2,0],[9E+09,1.01926,89.5581,9E+09,9E+09,9E+09]];
    PERS robtarget SPT54E:=[[-137.13,-21.49,129.92],[0.2715,-0.629431,0.285247,-0.669881],[0,1,-2,0],[9E+09,1.01926,89.5581,9E+09,9E+09,9E+09]];



    PERS pose SRT22:=[[0,0,0],[1,0,0,0]];


!!!!!!!!!!!!!!!!!!!!!!!!!!!!!!!!!!!!!!!!!!!!THUS ENDS THE ROBTARGETS!!!!!!!!!!!!!!!!!!!!!!!!!!!!!!!!!!!!!!!!!!!!!!!!!!!!!!!!!!!!!!!!!!!!!!!!
!!!!!!!!!!!!!!!!!!!!!!!!!!!!!!!!!!!!!!!!!!!!THUS BEGINS THE POSE!!!!!!!!!!!!!!!!!!!!!!!!!!!!!!!!!!!!!!!!!!!!!!!!!!!!!!!!!!!!!!!!!!!!!!!!

PERS pose SRG11:=[[0.0027771,-1.35965,-0.00526428],[1,0,0,0]];
PERS pose SRG12:=[[0.0155563,1.33756,0.0391846],[1,0,0,0]];
PERS pose SRT20:=[[-0.0445213,0.261669,-1.06805],[1,0,0,0]];
PERS pose SRT30:=[[-1.94688,-0.987652,0.0524292],[1,0,0,0]];
PERS pose SRT40:=[[-1.419,0.0980339,-0.772842],[1,0,0,0]];
PERS pose SRT50:=[[-0.175667,-0.945633,2.9303],[1,0,0,0]];
PERS pose SRAG100:=[[0,0,0],[1,0,0,0]];
PERS pose SRAH100:=[[0,0,0],[1,0,0,0]];
PERS pose SRG40:=[[0,0,0],[1,0,0,0]];
PERS pose SRH40:=[[0,0,0],[1,0,0,0]];
PERS pose SRG44:=[[0,0,0],[1,0,0,0]];
PERS pose SRG50:=[[0,0,0],[1,0,0,0]];
PERS pose SRH50:=[[0,0,0],[1,0,0,0]];
PERS pose SRH44:=[[0,0,0],[1,0,0,0]];
PERS pose SRH1:=[[0,0,0],[1,0,0,0]];
PERS pose SRH2:=[[0,0,0],[1,0,0,0]];
PERS pose SRG1:=[[0,0,0],[1,0,0,0]];
PERS pose SRG2:=[[0,0,0],[1,0,0,0]];
PERS pose SRAG101:=[[0,0,0],[1,0,0,0]];
PERS pose SRAH101:=[[0,0,0],[1,0,0,0]];
PERS pose SRT11:=[[0.123749,0.467068,0.0802765],[1,0,0,0]];
PERS pose SRR1Y:=[[0.0580521,0.414736,0.00358582],[1,0,0,0]];
PERS pose SRP1:=[[0.19075,0.00617599,0.94371],[1,0,0,0]];




  PERS pose SRPY:=[[0.0304394,0.00617599,-0.000946045],[1,0,0,0]];
  PERS pose SRPX:=[[0.19075,-0.00498199,-0.00491333],[1,0,0,0]];
  PERS pose poseBCG50:=[[-0.998383,0.100418,-7.68127],[1,0,0,0]];
  PERS pose SRG51:=[[0,0,0],[1,0,0,0]];
  PERS pose SRH51:=[[0,0,0],[1,0,0,0]];
  PERS pose T55:=[[1.35397,3.92874,-2.6429],[1,0,0,0]];
  PERS pose SRR11:=[[0.0487099,-5.06855,-5.73555],[1,0,0,0]];
  PERS pose SRG55:=[[0,0,0],[1,0,0,0]];
  PERS pose SRH55:=[[0,0,0],[1,0,0,0]];
  PERS pose SRG43:=[[0,0,0],[1,0,0,0]];
  PERS pose SRH43:=[[0,0,0],[1,0,0,0]];
  PERS pose SRT12X:=[[1.35397,0.0190773,-0.0292053],[1,0,0,0]];
  PERS pose SRG56:=[[0,0,0],[1,0,0,0]];
  PERS pose SRH56:=[[0,0,0],[1,0,0,0]];

  PERS pose SR_YZ_TEMP:=[[-0.00624895,-0.474304,-0.0861511],[1,0,0,0]];
  PERS pose SR_X_TEMP:=[[4.90775,-0.00191498,-0.0225525],[1,0,0,0]];




!!!!!!!!!!!!!!!!!!!!!!!!!!!!!!!!ASTUFFforSIP!!!!!!!!!!!!!!!!!!!!!!!!!!!!!!!!!!!!
!!!!DEFAULT VALUE OF A in the X is +18!!!!!

    PERS robtarget YA30S:=[[4.99,-324.826,583.669],[0.400321,-0.582805,-0.400834,0.582593],[-1,0,0,0],[9E+09,8.10884,-131.609,9E+09,9E+09,9E+09]];
    PERS robtarget YA30E:=[[4.99,-290.529,576.691],[0.400321,-0.582805,-0.400834,0.582593],[-1,0,0,0],[9E+09,8.10884,-131.609,9E+09,9E+09,9E+09]];
    PERS robtarget YA31S:=[[5,-494.369,994.058],[0.470811,-0.527513,-0.470884,0.527575],[-1,-1,0,0],[9E+09,9.82577,-131.326,9E+09,9E+09,9E+09]];
    PERS robtarget YA31E:=[[5,-400.027,980.052],[0.470811,-0.527513,-0.470884,0.527575],[-1,-1,0,0],[9E+09,9.82577,-131.326,9E+09,9E+09,9E+09]];
    PERS robtarget YA32S:=[[5,-334.398,493.223],[0.470811,-0.527513,-0.470884,0.527575],[-1,-1,0,0],[9E+09,-0.207107,-134.293,9E+09,9E+09,9E+09]];
    PERS robtarget YA32E:=[[5,-299.399,492.918],[0.470811,-0.527513,-0.470884,0.527575],[-1,-1,0,0],[9E+09,-0.207107,-134.293,9E+09,9E+09,9E+09]];
    PERS robtarget YA33S:=[[5,-328.035,414.295],[0.533623,-0.464168,-0.533363,0.464024],[-1,0,-1,0],[9E+09,-6.41779,-131.918,9E+09,9E+09,9E+09]];
    PERS robtarget YA33E:=[[4.99988,-293.515,420.072],[0.533623,-0.464168,-0.533363,0.464024],[0,-1,-1,0],[9E+09,-6.41779,-131.918,9E+09,9E+09,9E+09]];
    PERS robtarget YA34S:=[[5,-325.809,402.246],[0.537717,-0.459421,-0.537458,0.459274],[-1,0,-1,0],[9E+09,-7.68338,-131.683,9E+09,9E+09,9E+09]];
    PERS robtarget YA34E:=[[5,-291.452,408.924],[0.537717,-0.459421,-0.537458,0.459274],[-1,0,-1,0],[9E+09,-7.68338,-131.683,9E+09,9E+09,9E+09]];
    PERS robtarget YA325S:=[[18,-456.539,591.96],[0.542933,-0.452791,-0.543202,0.452919],[-1,-1,0,0],[9E+09,-13.34,-135,9E+09,9E+09,9E+09]];
    PERS robtarget YA325E:=[[18,-400.539,596.459],[0.542933,-0.452791,-0.543202,0.452919],[-1,-1,0,0],[9E+09,-13.34,-135,9E+09,9E+09,9E+09]];
    PERS robtarget YA39S:=[[5,-224.808,186.879],[0.639516,-0.3015,-0.639673,0.301555],[0,-1,-1,0],[9E+09,-28.169,-129.169,9E+09,9E+09,9E+09]];
    PERS robtarget YA39E:=[[5,-195.792,206.451],[0.639516,-0.3015,-0.639673,0.301555],[0,-1,-1,0],[9E+09,-28.169,-129.169,9E+09,9E+09,9E+09]];
    PERS robtarget YA38S:=[[5,-256.408,234.079],[0.633,-0.315232,-0.632899,0.315244],[0,-1,-1,0],[9E+09,-28.169,-129.169,9E+09,9E+09,9E+09]];
    PERS robtarget YA38E:=[[5,-227.392,253.651],[0.633,-0.315232,-0.632899,0.315244],[0,-1,-1,0],[9E+09,-28.169,-129.169,9E+09,9E+09,9E+09]];
    PERS robtarget YA37S:=[[5,-388.43,288.196],[0.587952,-0.393099,-0.58771,0.392915],[0,-1,-1,0],[9E+09,-24.9773,-129.477,9E+09,9E+09,9E+09]];
    PERS robtarget YA37E:=[[5,-300.732,318.648],[0.587952,-0.393099,-0.58771,0.392915],[0,-1,-1,0],[9E+09,-24.9773,-129.477,9E+09,9E+09,9E+09]];
    PERS robtarget YA36KS:=[[5,-466.184,453.465],[0.587952,-0.393099,-0.58771,0.392915],[0,-1,-1,0],[9E+09,-15.0841,-130.584,9E+09,9E+09,9E+09]];
    PERS robtarget YA36KE:=[[5,-373.626,473.494],[0.587952,-0.393099,-0.58771,0.392915],[0,-1,-1,0],[9E+09,-15.0841,-130.584,9E+09,9E+09,9E+09]];
    PERS robtarget YA35S:=[[5,-469.396,462.571],[0.587952,-0.393099,-0.58771,0.392915],[0,-1,-1,0],[9E+09,-14.6411,-130.641,9E+09,9E+09,9E+09]];
    PERS robtarget YA35E:=[[5,-376.664,482.105],[0.587952,-0.393099,-0.58771,0.392915],[0,-1,-1,0],[9E+09,-14.6411,-130.641,9E+09,9E+09,9E+09]];
    PERS robtarget YA36S:=[[5,-299.508,314.74],[0.587952,-0.393099,-0.58771,0.392915],[0,-1,-1,0],[9E+09,-17.7566,-130.257,9E+09,9E+09,9E+09]];
    PERS robtarget YA36E:=[[5,-267.172,328.134],[0.587952,-0.393099,-0.58771,0.392915],[0,-1,-1,0],[9E+09,-17.7566,-130.257,9E+09,9E+09,9E+09]];
    PERS robtarget YA33KS:=[[5,-520.13,813.206],[0.533623,-0.464168,-0.533363,0.464024],[-1,0,-1,0],[9E+09,0.918861,-133.419,9E+09,9E+09,9E+09]];
    PERS robtarget YA33KE:=[[5,-424.187,810.589],[0.533623,-0.464168,-0.533363,0.464024],[-1,0,-1,0],[9E+09,0.918861,-133.419,9E+09,9E+09,9E+09]];



    PERS robtarget A30air1:=[[585.02,-171.32,875.33],[0.678525,0.0623617,-0.709693,0.179035],[-1,2,-4,1],[9E+09,-4.8497,-134.909,9E+09,9E+09,9E+09]];
    PERS robtarget A30air2:=[[623.34,-168.87,991.22],[0.593636,0.334499,-0.574336,0.453703],[-1,2,-4,1],[9E+09,-4.84968,-134.909,9E+09,9E+09,9E+09]];
    PERS robtarget A30air3:=[[327.81,-490.47,907.80],[0.663233,0.140386,-0.672257,0.297468],[-1,2,-4,1],[9E+09,-4.84968,-134.909,9E+09,9E+09,9E+09]];
    PERS robtarget A30air10:=[[594.15,-159.02,869.61],[0.0797567,0.983892,0.150426,0.054494],[-1,2,-2,1],[9E+09,-4.84974,-134.909,9E+09,9E+09,9E+09]];
    PERS robtarget A30air11:=[[327.58,-346.63,841.21],[0.00514458,-0.986648,-0.155585,-0.047906],[-1,2,-2,1],[9E+09,-4.84968,-134.909,9E+09,9E+09,9E+09]];
    PERS robtarget A30air12:=[[371.47,-247.45,423.58],[0.190622,-0.967716,-0.15388,-0.0592667],[-1,2,-2,1],[9E+09,-4.84968,-134.909,9E+09,9E+09,9E+09]];
    PERS robtarget A39air1:=[[306.80,-429.51,348.64],[0.601772,-0.192288,-0.656352,0.41243],[-1,0,-1,0],[9E+09,0,-135,9E+09,9E+09,9E+09]];
    PERS robtarget A39air2:=[[306.80,-429.51,348.64],[0.601772,-0.192288,-0.656352,0.41243],[-1,0,-1,0],[9E+09,0,-135,9E+09,9E+09,9E+09]];
    PERS robtarget A39air3:=[[306.80,-429.51,348.64],[0.601772,-0.192288,-0.656352,0.41243],[-1,0,-1,0],[9E+09,0,-135,9E+09,9E+09,9E+09]];
    PERS robtarget A39air10:=[[364.93,-251.25,482.75],[0.00515267,-0.986648,-0.155581,-0.0479023],[-1,2,-2,1],[9E+09,0,-135,9E+09,9E+09,9E+09]];
    PERS robtarget A39air11:=[[364.93,-251.25,482.75],[0.00515291,-0.986648,-0.155581,-0.0479023],[-1,2,-2,1],[9E+09,0,-135,9E+09,9E+09,9E+09]];
    PERS robtarget A39air12:=[[364.93,-251.25,482.75],[0.00515291,-0.986648,-0.155581,-0.0479023],[-1,2,-2,1],[9E+09,0,-135,9E+09,9E+09,9E+09]];




    PERS robtarget XA39S:=[[151,-53.76,311.3],[0.000204649,1,-8.34711E-05,0.000184068],[0,2,-2,1],[9E+09,-28.169,-129.169,9E+09,9E+09,9E+09]];
    PERS robtarget XA39E:=[[121,-57.83,311.3],[0.00462409,-0.999989,8.48236E-05,-0.000184999],[0,2,-2,1],[9E+09,-28.169,-129.169,9E+09,9E+09,9E+09]];
    PERS robtarget XA33S:=[[151,-1.4,-344.34],[0.114211,-0.959087,-0.25724,-0.0305861],[-1,2,-2,1],[9E+09,-6.41779,-131.918,9E+09,9E+09,9E+09]];
    PERS robtarget XA33E:=[[121,-34.15,-52.36],[0.0117886,-0.965791,-0.259033,-0.00312085],[-1,2,-2,1],[9E+09,-6.41779,-131.918,9E+09,9E+09,9E+09]];
    PERS robtarget XA30S:=[[151,-27.57,-8.82],[0.000235893,-0.965864,-0.25905,-1.01904E-05],[-1,2,-2,1],[9E+09,8.10884,-131.609,9E+09,9E+09,9E+09]];
    PERS robtarget XA30E:=[[121,-38.04,69.43],[0.139073,0.955799,0.256344,-0.0373479],[-1,2,-2,1],[9E+09,8.10884,-131.609,9E+09,9E+09,9E+09]];
    PERS robtarget XA34S:=[[141,-66.88,-327.31],[0.000229182,-0.965864,-0.259052,-1.34677E-05],[-1,2,-2,1],[9E+09,-7.68338,-131.683,9E+09,9E+09,9E+09]];
    PERS robtarget XA34E:=[[121,-66.88,-327.31],[0.000229182,-0.965864,-0.259052,-1.34677E-05],[-1,2,-2,1],[9E+09,-7.68338,-131.683,9E+09,9E+09,9E+09]];
    PERS pose SRA30X:=[[-1.51614,0.00715256,-0.0129395],[1,0,0,0]];
    PERS pose SRA34X:=[[0,0,0],[1,0,0,0]];
    PERS pose SRA39X:=[[1.63543,0.0198669,0.0602722],[1,0,0,0]];
    PERS pose SRA33X:=[[0,0,0],[1,0,0,0]];



!!!!!!!!!!!!!!!!!!!!!!BSTUFFforSIP!!!!!!!!!!!!!!!!!!!!!!!!!!!!!!!!!!!!!!!!!
!!!!DEFAULT VALUE OF B in the X is -18!!!!!

    PERS robtarget YB30S:=[[-5,-324.826,583.669],[0.129142,0.695207,0.128921,0.695262],[-1,0,-3,0],[9E+09,8.10884,131.609,9E+09,9E+09,9E+09]];
    PERS robtarget YB30E:=[[-5,-290.529,576.691],[0.129142,0.695207,0.128921,0.695262],[-1,0,-3,0],[9E+09,8.10884,131.609,9E+09,9E+09,9E+09]];
    PERS robtarget YB31S:=[[-5,-494.369,994.058],[0.0401693,0.705998,0.0396681,0.70596],[-1,1,-3,0],[9E+09,9.82577,131.326,9E+09,9E+09,9E+09]];
    PERS robtarget YB31E:=[[-5,-400.027,980.052],[0.0401693,0.705998,0.0396681,0.70596],[-1,1,-3,0],[9E+09,9.82577,131.326,9E+09,9E+09,9E+09]];
    PERS robtarget YB32S:=[[-5,-334.398,493.223],[0.0401693,0.705998,0.0396681,0.70596],[-1,1,-3,0],[9E+09,-0.207107,134.293,9E+09,9E+09,9E+09]];
    PERS robtarget YB32E:=[[-5,-299.399,492.918],[0.0401693,0.705998,0.0396681,0.70596],[-1,1,-3,0],[9E+09,-0.207107,134.293,9E+09,9E+09,9E+09]];
    PERS robtarget YB33S:=[[-5,-328.035,414.295],[0.0487378,-0.705356,0.0499862,-0.705407],[-1,1,-3,0],[9E+09,-6.41779,131.918,9E+09,9E+09,9E+09]];
    PERS robtarget YB33E:=[[-5.00022,-293.515,420.072],[0.0487376,-0.705356,0.0499858,-0.705407],[-1,1,-3,0],[9E+09,-6.41779,131.918,9E+09,9E+09,9E+09]];
    PERS robtarget YB34S:=[[-5,-325.809,402.246],[0.0550159,-0.704884,0.0562635,-0.704945],[-1,1,-3,0],[9E+09,-7.68338,131.683,9E+09,9E+09,9E+09]];
    PERS robtarget YB34E:=[[-5,-291.452,408.924],[0.0550159,-0.704884,0.0562635,-0.704945],[-1,1,-3,0],[9E+09,-7.68338,131.683,9E+09,9E+09,9E+09]];
    PERS robtarget YB325S:=[[-18,-456.425,592.029],[0.00819136,0.707119,0.00799674,0.707002],[-1,1,-3,0],[9E+09,-13.34,135,9E+09,9E+09,9E+09]];
    PERS robtarget YB325E:=[[-18,-400.425,596.528],[0.00819136,0.707119,0.00799674,0.707002],[-1,1,-3,0],[9E+09,-13.34,135,9E+09,9E+09,9E+09]];
    PERS robtarget YB39S:=[[-5,-224.808,186.879],[0.239093,-0.665491,0.239369,-0.665326],[0,1,-3,0],[9E+09,-28.169,129.169,9E+09,9E+09,9E+09]];
    PERS robtarget YB39E:=[[-5,-195.792,206.451],[0.239093,-0.665491,0.239369,-0.665326],[0,1,-3,0],[9E+09,-28.169,129.169,9E+09,9E+09,9E+09]];
    PERS robtarget YB38S:=[[-5,-256.408,234.079],[0.224305,-0.670601,0.224383,-0.670547],[0,1,-3,0],[9E+09,-28.169,129.169,9E+09,9E+09,9E+09]];
    PERS robtarget YB38E:=[[-5,-227.392,253.651],[0.224305,-0.670601,0.224383,-0.670547],[0,1,-3,0],[9E+09,-28.169,129.169,9E+09,9E+09,9E+09]];
    PERS robtarget YB37S:=[[-4.99,-388.43,288.196],[0.137592,-0.693364,0.138822,-0.693573],[-1,1,-3,0],[9E+09,-24.9773,129.477,9E+09,9E+09,9E+09]];
    PERS robtarget YB37E:=[[-4.99,-300.732,318.648],[0.137592,-0.693364,0.138822,-0.693573],[-1,1,-3,0],[9E+09,-24.9773,129.477,9E+09,9E+09,9E+09]];
    PERS robtarget YB36KS:=[[-4.99,-466.184,453.465],[0.137592,-0.693364,0.138822,-0.693573],[-1,1,-3,0],[9E+09,-15.0841,130.584,9E+09,9E+09,9E+09]];
    PERS robtarget YB36KE:=[[-4.99,-373.626,473.494],[0.137592,-0.693364,0.138822,-0.693573],[-1,1,-3,0],[9E+09,-15.0841,130.584,9E+09,9E+09,9E+09]];
    PERS robtarget YB35S:=[[-4.99,-469.396,462.571],[0.137592,-0.693364,0.138822,-0.693573],[-1,1,-3,0],[9E+09,-14.6411,130.641,9E+09,9E+09,9E+09]];
    PERS robtarget YB35E:=[[-4.99,-376.664,482.105],[0.137592,-0.693364,0.138822,-0.693573],[-1,1,-3,0],[9E+09,-14.6411,130.641,9E+09,9E+09,9E+09]];
    PERS robtarget YB36S:=[[-4.99,-299.508,314.74],[0.137592,-0.693364,0.138822,-0.693573],[-1,1,-3,0],[9E+09,-17.7566,130.257,9E+09,9E+09,9E+09]];
    PERS robtarget YB36E:=[[-4.99,-267.172,328.134],[0.137592,-0.693364,0.138822,-0.693573],[-1,1,-3,0],[9E+09,-17.7566,130.257,9E+09,9E+09,9E+09]];
    PERS robtarget YB33KS:=[[-5,-520.13,813.206],[0.0487378,-0.705356,0.0499862,-0.705407],[-1,1,-3,0],[9E+09,0.918861,133.419,9E+09,9E+09,9E+09]];
    PERS robtarget YB33KE:=[[-5,-424.187,810.589],[0.0487378,-0.705356,0.0499862,-0.705407],[-1,1,-3,0],[9E+09,0.918861,133.419,9E+09,9E+09,9E+09]];




    PERS robtarget B30air1:=[[-504.23,-214.11,666.64],[0.174665,0.714629,-0.148749,0.660811],[-1,0,-3,0],[9E+09,-5.48905,135.061,9E+09,9E+09,9E+09]];
    PERS robtarget B30air2:=[[-493.15,-367.93,1057.05],[0.0545492,0.726886,-0.0369722,0.68359],[-1,0,-3,0],[9E+09,-5.489,135.061,9E+09,9E+09,9E+09]];
    PERS robtarget B30air3:=[[-201.11,-567.29,927.35],[0.234652,0.678877,-0.198792,0.666743],[-1,0,-3,0],[9E+09,-5.48907,135.061,9E+09,9E+09,9E+09]];
    PERS robtarget B30air10:=[[-494.00,-330.26,1053.17],[0.0572997,-0.0428609,-0.997168,-0.023179],[-1,0,-1,0],[9E+09,-5.48903,135.061,9E+09,9E+09,9E+09]];
    PERS robtarget B30air11:=[[-389.05,-325.33,767.75],[0.0573001,-0.0428617,-0.997168,-0.0231749],[-1,1,-1,0],[9E+09,-5.48905,135.061,9E+09,9E+09,9E+09]];
    PERS robtarget B30air12:=[[-389.04,-325.32,767.75],[0.0573003,-0.0428623,-0.997168,-0.0231752],[-1,1,-1,0],[9E+09,-5.48903,135.061,9E+09,9E+09,9E+09]];


    PERS robtarget B39air1:=[[-323.48,-348.44,373.29],[0.122788,0.72187,-0.311157,0.605812],[-1,1,-3,0],[9E+09,0,135,9E+09,9E+09,9E+09]];
    PERS robtarget B39air2:=[[-279.95,-312.15,117.83],[0.0211591,0.670472,-0.195567,0.715384],[0,1,-3,0],[9E+09,0,135,9E+09,9E+09,9E+09]];
    PERS robtarget B39air3:=[[-323.48,-348.44,373.29],[0.122788,0.72187,-0.311157,0.605812],[-1,1,-3,0],[9E+09,0,135,9E+09,9E+09,9E+09]];
    PERS robtarget B39air10:=[[-434.18,-117.02,196.36],[0.0372703,-0.167052,-0.937721,-0.302301],[0,1,-1,0],[9E+09,0,135,9E+09,9E+09,9E+09]];
    PERS robtarget B39air11:=[[-434.18,-117.02,196.36],[0.0372703,-0.167052,-0.93772,-0.302301],[0,1,-1,0],[9E+09,0,135,9E+09,9E+09,9E+09]];
    PERS robtarget B39air12:=[[-434.18,-117.02,196.36],[0.037271,-0.167052,-0.93772,-0.302303],[0,1,-1,0],[9E+09,-5.48905,135.061,9E+09,9E+09,9E+09]];

    PERS robtarget XB39S:=[[-151,-52.98,326.2],[2.8716E-05,-0.00039622,-1,5.17092E-05],[0,1,-1,0],[9E+09,-28.169,129.169,9E+09,9E+09,9E+09]];
    PERS robtarget XB39E:=[[-121,-60.59,313.79],[3.83994E-06,-0.000396945,-0.998119,0.0613129],[0,1,-1,0],[9E+09,-28.169,129.169,9E+09,9E+09,9E+09]];
    PERS robtarget XB33S:=[[-151,23.06,-394.59],[7.92389E-05,-0.000185338,-0.989356,-0.145515],[-1,1,-1,0],[9E+09,-6.41779,131.918,9E+09,9E+09,9E+09]];
    PERS robtarget XB33E:=[[-121,-25.54,-63.96],[5.87928E-05,-0.000190698,-0.998771,-0.0495659],[-1,1,-1,0],[9E+09,-6.41779,131.918,9E+09,9E+09,9E+09]];
    PERS robtarget XB30S:=[[-151,-27.1,-4.74],[0.00031804,-0.000205712,-1,-9.57148E-05],[-1,0,-1,0],[9E+09,8.10884,131.609,9E+09,9E+09,9E+09]];
    PERS robtarget XB30E:=[[-121,-23.86,74.64],[0.000296319,-0.000232285,-0.995746,0.0921449],[-1,1,-1,0],[9E+09,8.10884,131.609,9E+09,9E+09,9E+09]];
    PERS robtarget XB34S:=[[-141,-60.01,-301.76],[5.17653E-05,-0.000194982,-1,-0.000245567],[-1,1,-1,0],[9E+09,-7.68338,131.683,9E+09,9E+09,9E+09]];
    PERS robtarget XB34E:=[[-121,-60.01,-301.76],[5.17653E-05,-0.000194982,-1,-0.000245567],[-1,1,-1,0],[9E+09,-7.68338,131.683,9E+09,9E+09,9E+09]];
    PERS pose SRB30X:=[[-1.73971,0.00458717,-0.0296555],[1,0,0,0]];
    PERS pose SRB34X:=[[0,0,0],[1,0,0,0]];
    PERS pose SRB39X:=[[-3.30756,0.00440979,0.0306091],[1,0,0,0]];
    PERS pose SRB33X:=[[-2.60141,-0.00635147,0.0080986],[1,0,0,0]];



!!!!!!!!!!!!!!!!!!!!!!!!!!!!!!!!GSTUFFforSIP!!!!!!!!!!!!!!!!!!!!!!!!!!!!!!!!!!!!
!!!!DEFAULT VALUE OF G in the X is - 18!!!!!

    PERS robtarget YG29S:=[[-5,-58.2555,703.15],[0.15894,0.689021,0.15928,0.688925],[-1,0,-2,0],[9E+09,-18.2042,49.7958,9E+09,9E+09,9E+09]];
    PERS robtarget YG29E:=[[-5,-90.4732,716.825],[0.15894,0.689021,0.15928,0.688925],[-1,0,-2,0],[9E+09,-18.2042,49.7958,9E+09,9E+09,9E+09]];
    PERS robtarget YG27S:=[[-5,-146.086,1157.84],[0.0801795,0.70252,0.0798257,0.702613],[-1,0,-2,0],[9E+09,-20,50,9E+09,9E+09,9E+09]];
    PERS robtarget YG27E:=[[-5,-164.465,1183.19],[0.0801795,0.70252,0.0798257,0.702613],[-1,0,-2,0],[9E+09,-20,50,9E+09,9E+09,9E+09]];
    PERS robtarget YG25S:=[[-5,-100.05,578.503],[0.0801795,0.70252,0.0798257,0.702613],[-1,0,-2,0],[9E+09,-8.96447,48.5355,9E+09,9E+09,9E+09]];
    PERS robtarget YG25E:=[[-5,-134.22,586.078],[0.0801795,0.70252,0.0798257,0.702613],[-1,0,-2,0],[9E+09,-8.96447,48.5355,9E+09,9E+09,9E+09]];
    PERS robtarget YG23S:=[[-5,-207.941,985.197],[0.0801795,0.70252,0.0798257,0.702613],[-1,0,-2,0],[9E+09,-10.6921,48.8079,9E+09,9E+09,9E+09]];
    PERS robtarget YG23E:=[[-5,-230.03,1000.22],[0.0801795,0.70252,0.0798257,0.702613],[-1,0,-2,0],[9E+09,-10.6921,48.8079,9E+09,9E+09,9E+09]];
    PERS robtarget YG0S:=[[-5,-114.202,449.077],[0.00333448,0.707035,0.00299418,0.707165],[-1,0,-2,0],[9E+09,0.207107,45.7071,9E+09,9E+09,9E+09]];
    PERS robtarget YG0E:=[[-5.00011,-149.201,449.382],[0.00333469,0.707035,0.00299401,0.707165],[-1,0,-2,0],[9E+09,0.207107,45.7071,9E+09,9E+09,9E+09]];
    PERS robtarget YG19S:=[[-5.03,-82.8063,258.489],[0.130951,-0.694906,0.130628,-0.694906],[-1,0,-2,0],[9E+09,14.1988,49.3012,9E+09,9E+09,9E+09]];
    PERS robtarget YG19E:=[[-5.03,-115.998,247.384],[0.130951,-0.694906,0.130628,-0.694906],[-1,0,-2,0],[9E+09,14.1988,49.3012,9E+09,9E+09,9E+09]];
    PERS robtarget YG18S:=[[-5.01,-87.1447,271.884],[0.134872,-0.694026,0.13526,-0.694148],[-1,0,-2,0],[9E+09,13.3167,49.1833,9E+09,9E+09,9E+09]];
    PERS robtarget YG18E:=[[-5.01,-120.525,261.36],[0.134872,-0.694026,0.13526,-0.694148],[-1,0,-2,0],[9E+09,13.3167,49.1833,9E+09,9E+09,9E+09]];
    PERS robtarget YG16S:=[[-5,-189.098,442.522],[0.067801,-0.703752,0.0681279,-0.703915],[-1,0,-2,0],[9E+09,14.1988,49.3012,9E+09,9E+09,9E+09]];
    PERS robtarget YG16E:=[[-5,-209.998,423.484],[0.067801,-0.703752,0.0681279,-0.703915],[-1,0,-2,0],[9E+09,14.1988,49.3012,9E+09,9E+09,9E+09]];
    PERS robtarget YG15S:=[[-5,-107.333,359.469],[0.067801,-0.703752,0.0681279,-0.703915],[-1,0,-2,0],[9E+09,5.58452,47.9155,9E+09,9E+09,9E+09]];
    PERS robtarget YG15E:=[[-5.00035,-141.948,354.295],[0.0678008,-0.703752,0.0681281,-0.703915],[-1,0,-2,0],[9E+09,5.58452,47.9155,9E+09,9E+09,9E+09]];
    PERS robtarget YG10S:=[[-5,-229.829,621.094],[0.067801,-0.703752,0.0681279,-0.703915],[-1,0,-2,0],[9E+09,4.76139,47.7386,9E+09,9E+09,9E+09]];
    PERS robtarget YG10E:=[[-5,-253.315,613.262],[0.067801,-0.703752,0.0681279,-0.703915],[-1,0,-2,0],[9E+09,4.76139,47.7386,9E+09,9E+09,9E+09]];
    PERS robtarget YG21S:=[[-5,-114.102,460.923],[0.00315908,0.707036,0.00281907,0.707165],[-1,0,-2,0],[9E+09,-0.207107,45.7071,9E+09,9E+09,9E+09]];
    PERS robtarget YG21E:=[[-5.00011,-149.101,460.618],[0.00315932,0.707036,0.00281869,0.707165],[-1,0,-2,0],[9E+09,-0.207107,45.7071,9E+09,9E+09,9E+09]];
    PERS robtarget YG15KS:=[[-5,-228.715,612.829],[0.067801,-0.703752,0.0681279,-0.703915],[-1,0,-2,0],[9E+09,1.03,45,9E+09,9E+09,9E+09]];
    PERS robtarget YG15KE:=[[-5,-252.131,604.479],[0.067801,-0.703752,0.0681279,-0.703915],[-1,0,-2,0],[9E+09,1.03,45,9E+09,9E+09,9E+09]];
    PERS robtarget YG21KS:=[[-5,-236.237,804.213],[0.00315908,0.707036,0.00281907,0.707165],[-1,0,-2,0],[9E+09,-1.62917,46.8708,9E+09,9E+09,9E+09]];
    PERS robtarget YG21KE:=[[-5,-260.125,807.876],[0.00315908,0.707036,0.00281907,0.707165],[-1,0,-2,0],[9E+09,-1.62917,46.8708,9E+09,9E+09,9E+09]];



    PERS robtarget G19air1:=[[-249.66,31.69,426.64],[0.360781,-0.61592,0.272934,-0.644971],[-1,0,-1,0],[9E+09,0,45,9E+09,9E+09,9E+09]];
    PERS robtarget G19air2:=[[-407.16,43.62,424.98],[0.121877,-0.624623,-0.148501,-0.756926],[-1,0,-2,0],[9E+09,0,45,9E+09,9E+09,9E+09]];
    PERS robtarget G19air3:=[[-337.34,-83.17,634.9],[0.0875438,0.658657,0.141506,0.733815],[-1,0,-2,0],[9E+09,0,45,9E+09,9E+09,9E+09]];
    PERS robtarget G19air10:=[[-545,-455.08,338.98],[0.183295,0.0846019,-0.94126,-0.270696],[0,0,1,0],[9E+09,0,45,9E+09,9E+09,9E+09]];
    PERS robtarget G19air11:=[[-418.41,-219.04,252.70],[0.0807707,0.090812,-0.968993,-0.215137],[-1,0,1,0],[9E+09,2.3391E-05,45,9E+09,9E+09,9E+09]];
    PERS robtarget G19air12:=[[505.89,-331.92,460.47],[0.0666954,-0.996457,-0.0305737,-0.0411239],[-1,0,-1,0],[9E+09,-7.78641E-06,-45,9E+09,9E+09,9E+09]];
    PERS robtarget G29air1:=[[-345.57,13.71,693.64],[0.280425,-0.644333,0.196707,-0.683743],[-1,0,-1,0],[9E+09,0,45,9E+09,9E+09,9E+09]];
    PERS robtarget G29air2:=[[-192.07,28.01,707.93],[0.280424,-0.644333,0.196707,-0.683743],[-1,0,-1,0],[9E+09,0,45,9E+09,9E+09,9E+09]];
    PERS robtarget G29air3:=[[-192.07,28.01,707.93],[0.280424,-0.644333,0.196707,-0.683743],[-1,0,-1,0],[9E+09,0,45,9E+09,9E+09,9E+09]];
    PERS robtarget G29air10:=[[-484.04,-133.98,1285.11],[0.00144517,-0.0082516,-0.844927,-0.534817],[-1,-1,1,0],[9E+09,-26.7991,50.7009,9E+09,9E+09,9E+09]];
    PERS robtarget G29air11:=[[-274.46,-298.84,357.69],[0.0400899,0.219433,-0.926836,0.302022],[-1,0,0,0],[9E+09,0,45,9E+09,9E+09,9E+09]];
    PERS robtarget G29air12:=[[-328.96,-278.4,1041],[0.128348,0.200172,-0.950789,0.198644],[-1,0,0,0],[9E+09,0,45,9E+09,9E+09,9E+09]];

    PERS robtarget XG19S:=[[-151,-53.67,329.08],[0.000262748,-0.00032762,1,0.000156863],[-1,0,0,0],[9E+09,14.1988,49.3012,9E+09,9E+09,9E+09]];
    PERS robtarget XG19E:=[[-120.8,-54.87,303.73],[0.000251312,-0.000335351,0.999459,-0.0328896],[-1,0,0,0],[9E+09,14.1988,49.3012,9E+09,9E+09,9E+09]];
    PERS robtarget XG21S:=[[-141,-39.02,-298.96],[1.78506E-05,-0.000207247,1,-0.000110213],[-1,0,0,0],[9E+09,-0.207107,45.7071,9E+09,9E+09,9E+09]];
    PERS robtarget XG21E:=[[-121,-39.02,-298.96],[1.78506E-05,-0.000207247,1,-0.000110213],[-1,0,0,0],[9E+09,-0.207107,45.7071,9E+09,9E+09,9E+09]];
    PERS robtarget XG0S:=[[-151,17.72,-298.19],[3.77814E-05,-0.00020441,0.995216,0.0977038],[-1,0,0,0],[9E+09,0.207107,45.7071,9E+09,9E+09,9E+09]];
    PERS robtarget XG0E:=[[-120.8,-11.33,-40.59],[1.61491E-05,-0.000206777,0.999994,-0.00359837],[-1,0,0,0],[9E+09,0.207107,45.7071,9E+09,9E+09,9E+09]];
    PERS robtarget XG29S:=[[-151,-47.02,-193.16],[0.00364056,-0.00441893,-0.0159999,-0.999856],[-1,-1,2,0],[9E+09,-18.2042,49.7958,9E+09,9E+09,9E+09]];
    PERS robtarget XG29E:=[[-120.8,-42.11,-288.2],[5.55738E-05,-0.000199481,0.982027,0.188743],[-1,0,0,0],[9E+09,-18.2042,49.7958,9E+09,9E+09,9E+09]];
    PERS pose SRG29X:=[[0.0123672,-0.00711823,-0.0197144],[1,0,0,0]];
    PERS pose SRG0X:=[[-1.08789,0.00152683,-0.0116119],[1,0,0,0]];
    PERS pose SRG19X:=[[-2.27755,0.0210152,-0.0202026],[1,0,0,0]];
    PERS pose SRG21X:=[[0,0,0],[1,0,0,0]];


          !!!!!!!!!!!!!!!!HSTUFFforSIP!!!!!!!!!!!!!!!!!!!!!!
!!!!DEFAULT VALUE OF H in the X is +18!!!!!

    PERS robtarget YH29S:=[[5,-58.2555,703.15],[0.655366,-0.265636,-0.655379,0.26535],[-1,1,-3,0],[9E+09,-18.2042,-49.7958,9E+09,9E+09,9E+09]];
    PERS robtarget YH29E:=[[5,-90.4732,716.825],[0.655366,-0.265636,-0.655379,0.26535],[-1,1,-3,0],[9E+09,-18.2042,-49.7958,9E+09,9E+09,9E+09]];
    PERS robtarget YH27S:=[[5,-146.086,1157.84],[0.655588,-0.26514,-0.655537,0.264911],[-1,1,-3,0],[9E+09,-20,-50,9E+09,9E+09,9E+09]];
    PERS robtarget YH27E:=[[5,-162.465,1183.19],[0.655588,-0.26514,-0.655537,0.264911],[-1,1,-3,0],[9E+09,-20,-50,9E+09,9E+09,9E+09]];
    PERS robtarget YH25S:=[[5,-100.05,578.503],[0.655588,-0.26514,-0.655537,0.264911],[-1,1,-3,0],[9E+09,-8.96447,-48.5355,9E+09,9E+09,9E+09]];
    PERS robtarget YH25E:=[[5,-134.22,586.078],[0.655588,-0.26514,-0.655537,0.264911],[-1,1,-3,0],[9E+09,-8.96447,-48.5355,9E+09,9E+09,9E+09]];
    PERS robtarget YH23S:=[[5,-207.941,985.197],[0.655588,-0.26514,-0.655537,0.264911],[-1,1,-3,0],[9E+09,-10.6921,-48.8079,9E+09,9E+09,9E+09]];
    PERS robtarget YH23E:=[[5,-228.03,1000.22],[0.655588,-0.26514,-0.655537,0.264911],[-1,1,-3,0],[9E+09,-10.6921,-48.8079,9E+09,9E+09,9E+09]];
    PERS robtarget YH0S:=[[5,-114.202,449.077],[0.655588,-0.265138,-0.655537,0.26491],[-1,1,-3,0],[9E+09,0.207107,-45.7071,9E+09,9E+09,9E+09]];
    PERS robtarget YH0E:=[[5.00016,-149.201,449.382],[0.655588,-0.265138,-0.655537,0.26491],[-1,1,-3,0],[9E+09,0.207107,-45.7071,9E+09,9E+09,9E+09]];


    PERS robtarget YH19S:=[[5.01,-82.8063,258.489],[0.701394,-0.0885962,-0.701664,0.0886789],[-1,1,-3,0],[9E+09,14.1988,-49.3012,9E+09,9E+09,9E+09]];
    PERS robtarget YH19E:=[[5.01,-115.998,247.384],[0.701394,-0.0885962,-0.701664,0.0886789],[-1,1,-3,0],[9E+09,14.1988,-49.3012,9E+09,9E+09,9E+09]];
    PERS robtarget YH18S:=[[5.01,-87.1447,271.884],[0.701649,-0.0886661,-0.701413,0.0885831],[-1,1,-3,0],[9E+09,13.3167,-49.1833,9E+09,9E+09,9E+09]];
    PERS robtarget YH18E:=[[5.01,-120.525,261.36],[0.701649,-0.0886661,-0.701413,0.0885831],[-1,1,-3,0],[9E+09,13.3167,-49.1833,9E+09,9E+09,9E+09]];
    PERS robtarget YH16S:=[[5,-189.098,442.522],[0.655588,-0.265137,-0.655538,0.264909],[-1,1,-3,0],[9E+09,14.1988,-49.3012,9E+09,9E+09,9E+09]];
    PERS robtarget YH16E:=[[5,-207.998,423.484],[0.655588,-0.265137,-0.655538,0.264909],[-1,1,-3,0],[9E+09,14.1988,-49.3012,9E+09,9E+09,9E+09]];
    PERS robtarget YH15S:=[[5,-107.333,359.469],[0.655588,-0.265137,-0.655538,0.264909],[-1,1,-3,0],[9E+09,5.58452,-47.9155,9E+09,9E+09,9E+09]];
    PERS robtarget YH15E:=[[5.00013,-141.948,354.295],[0.655588,-0.265137,-0.655538,0.264909],[-1,1,-3,0],[9E+09,5.58452,-47.9155,9E+09,9E+09,9E+09]];
    PERS robtarget YH10S:=[[5,-229.829,621.094],[0.655588,-0.265137,-0.655538,0.264909],[-1,1,-3,0],[9E+09,4.76139,-47.7386,9E+09,9E+09,9E+09]];
    PERS robtarget YH10E:=[[5,-251.315,613.262],[0.655588,-0.265137,-0.655538,0.264909],[-1,1,-3,0],[9E+09,4.76139,-47.7386,9E+09,9E+09,9E+09]];
    PERS robtarget YH21S:=[[5,-114.102,460.923],[0.655589,-0.265135,-0.655538,0.264908],[-1,1,-3,0],[9E+09,-0.207107,-45.7071,9E+09,9E+09,9E+09]];
    PERS robtarget YH21E:=[[5.00035,-149.101,460.618],[0.655589,-0.265135,-0.655538,0.264908],[-1,1,-3,0],[9E+09,-0.207107,-45.7071,9E+09,9E+09,9E+09]];
    PERS robtarget YH15KS:=[[5,-228.715,612.829],[0.655588,-0.265137,-0.655538,0.264909],[-1,1,-3,0],[9E+09,1.03,-45,9E+09,9E+09,9E+09]];
    PERS robtarget YH15KE:=[[5,-250.131,604.479],[0.655588,-0.265137,-0.655538,0.264909],[-1,1,-3,0],[9E+09,1.03,-45,9E+09,9E+09,9E+09]];
    PERS robtarget YH21KS:=[[5,-236.237,804.213],[0.655589,-0.265135,-0.655538,0.264908],[-1,1,-3,0],[9E+09,-1.62917,-46.8708,9E+09,9E+09,9E+09]];
    PERS robtarget YH21KE:=[[5,-258.125,807.876],[0.655589,-0.265135,-0.655538,0.264908],[-1,1,-3,0],[9E+09,-1.62917,-46.8708,9E+09,9E+09,9E+09]];


    PERS robtarget XH19S:=[[151,-52.55,358.06],[0.000101309,-1,0.000358162,9.67526E-05],[-1,0,-1,0],[9E+09,14.1988,-49.3012,9E+09,9E+09,9E+09]];
    PERS robtarget XH19E:=[[120.8,-58.15,313.55],[0.0750769,0.997178,-0.000364188,-6.95723E-05],[-1,1,-1,0],[9E+09,14.1988,-49.3012,9E+09,9E+09,9E+09]];
    PERS robtarget XH21S:=[[141,-33.64,-269.42],[0.000224467,1,-0.00029816,-0.000155511],[-1,1,-1,0],[9E+09,-0.207107,-45.7071,9E+09,9E+09,9E+09]];
    PERS robtarget XH21E:=[[121,-33.64,-269.42],[0.000224467,1,-0.00029816,-0.000155511],[-1,1,-1,0],[9E+09,-0.207107,-45.7071,9E+09,9E+09,9E+09]];
    PERS robtarget XH29S:=[[151,-48.54,-319.96],[3.2876E-05,-1,9.3793E-05,-0.000104989],[-1,1,-1,0],[9E+09,-18.2042,-49.7958,9E+09,9E+09,9E+09]];
    PERS robtarget XH29E:=[[120.8,-43.22,-319.96],[0.139406,-0.990235,0.00010758,-9.06353E-05],[-1,1,-1,0],[9E+09,-18.2042,-49.7958,9E+09,9E+09,9E+09]];
    PERS robtarget XH0S:=[[151,7.5,-269.42],[0.0788113,-0.996889,0.000284967,0.000178685],[-1,1,-1,0],[9E+09,0.207107,-45.7071,9E+09,9E+09,9E+09]];
    PERS robtarget XH0E:=[[120.8,-3.48,-15.26],[0.0329366,-0.999457,0.000293029,0.000165777],[-1,1,-1,0],[9E+09,0.207107,-45.7071,9E+09,9E+09,9E+09]];
    PERS pose SRH29X:=[[2.62572,-0.000324249,0.0204468],[1,0,0,0]];
    PERS pose SRH0X:=[[0.137779,0.0210199,0.0227432],[1,0,0,0]];
    PERS pose SRH19X:=[[-0.187057,-1.14441E-05,0.0199585],[1,0,0,0]];
    PERS pose SRH21X:=[[0,0,0],[1,0,0,0]];


    PERS robtarget H19air1:=[[679.25,-204.99,279.23],[0.587637,-0.237989,-0.773121,0.0181478],[-1,1,-2,0],[9E+09,0,-45,9E+09,9E+09,9E+09]];
    PERS robtarget H19air2:=[[679.25,-205.00,279.23],[0.58764,-0.237989,-0.773119,0.0181527],[-1,1,-2,0],[9E+09,2.3391E-05,-45,9E+09,9E+09,9E+09]];
    PERS robtarget H19air3:=[[277.83,-12.76,658.85],[0.723742,-0.0971594,-0.678098,0.0833208],[-1,1,-3,0],[9E+09,2.3391E-05,-45,9E+09,9E+09,9E+09]];
    PERS robtarget H19air10:=[[466.90,-237.60,593.85],[0.0785752,-0.993933,-0.031119,-0.070394],[-1,0,-1,0],[9E+09,0,-45,9E+09,9E+09,9E+09]];
    PERS robtarget H19air11:=[[386.84,-158.20,163.67],[0.264082,-0.961425,-0.0437994,-0.0632873],[0,0,-1,0],[9E+09,2.3391E-05,-45,9E+09,9E+09,9E+09]];
    PERS robtarget H19air12:=[[466.9,-237.6,593.85],[0.0785751,-0.993933,-0.0311191,-0.0703939],[-1,0,-1,0],[9E+09,0,-45,9E+09,9E+09,9E+09]];
    PERS robtarget H29air1:=[[387.66,34.32,760.81],[0.679544,-0.392394,-0.615068,0.0770624],[-1,1,-3,0],[9E+09,0,-45,9E+09,9E+09,9E+09]];
    PERS robtarget H29air2:=[[312.79,116.60,1033.81],[0.505745,-0.365251,-0.765628,0.156936],[-1,1,-3,0],[9E+09,-21.5,-50.0002,9E+09,9E+09,9E+09]];
    PERS robtarget H29air3:=[[387.66,34.32,760.81],[0.679544,-0.392394,-0.615068,0.0770624],[-1,1,-3,0],[9E+09,0,-45,9E+09,9E+09,9E+09]];
    PERS robtarget H29air10:=[[469.77,-61.48,1151.25],[0.236494,0.969947,0.0278606,0.0499777],[-1,1,-1,0],[9E+09,-21.5019,-50.0004,9E+09,9E+09,9E+09]];
    PERS robtarget H29air11:=[[375.59,-231.13,1059.75],[0.236492,0.969948,0.0278585,0.0499781],[-1,1,-1,0],[9E+09,-21.5019,-50.0005,9E+09,9E+09,9E+09]];
    PERS robtarget H29air12:=[[500,-336.51,649.64],[0.236488,0.969949,0.0278585,0.0499782],[-1,1,-1,0],[9E+09,0,-45,9E+09,9E+09,9E+09]];


    PERS robtarget F90airBETWEENXB30_34:=[[-315.58,-237.68,582.73],[0.000305905,-0.000201023,-0.999764,0.0217172],[-1,1,-1,0],[9E+09,0,135,9E+09,9E+09,9E+09]];
    PERS robtarget F90airBETWEENX29_0G:=[[-244.68,-207.48,614.12],[8.93859E-06,-0.000207923,0.99976,-0.0219144],[-1,0,0,0],[9E+09,0,45,9E+09,9E+09,9E+09]];
    PERS robtarget F90airBETWEENX19_21G:=[[-256.78,-213.61,292.41],[0.0424114,0.0870616,-0.995227,-0.0120583],[-1,0,0,0],[9E+09,0,45,9E+09,9E+09,9E+09]];
    PERS robtarget F90airBETWEENX19_21H:=[[265.79,-206.68,446.05],[0.0884887,-0.993446,-0.0353398,-0.0631317],[-1,1,-1,0],[9E+09,0,-45,9E+09,9E+09,9E+09]];

   !!!!!!!!!!!!!!!!!!!!        L STUFF FOR SIP   !!!!!!!!!!!!!!!!!!!!

!!!!DEFAULT VALUE OF L in the X is +8!!!!!

    PERS robtarget YL41S:=[[0,-113.919,467.621],[0.527354,0.470863,-0.527632,-0.470947],[-1,1,-1,0],[9E+09,-0.275255,46.2247,9E+09,9E+09,9E+09]];
    PERS robtarget YL41E:=[[0,-148.907,468.537],[0.527354,0.470863,-0.527632,-0.470947],[-1,1,-1,0],[9E+09,-0.275255,46.2247,9E+09,9E+09,9E+09]];
    PERS robtarget YL42S:=[[0.01,-110.263,518.104],[0.545581,0.449595,-0.545878,-0.449692],[-1,1,-1,0],[9E+09,-3.95049,47.5495,9E+09,9E+09,9E+09]];
    PERS robtarget YL42E:=[[0.01,-145.038,522.066],[0.545581,0.449595,-0.545878,-0.449692],[-1,1,-1,0],[9E+09,-3.95049,47.5495,9E+09,9E+09,9E+09]];
    PERS robtarget YL46S:=[[0.01,-100.139,577.971],[0.564756,0.425495,-0.564713,-0.425563],[-1,1,-1,0],[9E+09,-8.96447,48.5355,9E+09,9E+09,9E+09]];
    PERS robtarget YL46E:=[[0.01,-134.31,585.547],[0.564756,0.425495,-0.564713,-0.425563],[-1,1,-1,0],[9E+09,-8.96447,48.5355,9E+09,9E+09,9E+09]];
    PERS robtarget YL45S:=[[0,-102.234,568.136],[0.561097,0.430232,-0.561232,-0.43022],[-1,1,-1,0],[9E+09,-8.10884,48.3912,9E+09,9E+09,9E+09]];
    PERS robtarget YL45E:=[[0,-136.532,575.114],[0.561097,0.430232,-0.561232,-0.43022],[-1,1,-1,0],[9E+09,-8.10884,48.3912,9E+09,9E+09,9E+09]];
    PERS robtarget YL47S:=[[0,-90.0267,617.353],[0.577685,0.40797,-0.577373,-0.408021],[-1,1,-1,0],[9E+09,-12.438,49.062,9E+09,9E+09,9E+09]];
    PERS robtarget YL47E:=[[0,-123.585,627.294],[0.577685,0.40797,-0.577373,-0.408021],[-1,1,-1,0],[9E+09,-12.438,49.062,9E+09,9E+09,9E+09]];
    PERS robtarget YL48S:=[[0,-73.7314,665.293],[0.593176,0.385137,-0.592906,-0.385063],[-1,1,-1,0],[9E+09,-16.8632,49.6368,9E+09,9E+09,9E+09]];
    PERS robtarget YL48E:=[[0,-106.296,678.12],[0.593176,0.385137,-0.592906,-0.385063],[-1,1,-1,0],[9E+09,-16.8632,49.6368,9E+09,9E+09,9E+09]];
    PERS robtarget YL49S:=[[0,-66.5915,682.424],[0.604333,0.366803,-0.60467,-0.366895],[-1,1,-1,0],[9E+09,-18.2042,49.7958,9E+09,9E+09,9E+09]];
    PERS robtarget YL49E:=[[0,-98.8091,696.099],[0.604333,0.366803,-0.60467,-0.366895],[-1,1,-1,0],[9E+09,-18.2042,49.7958,9E+09,9E+09,9E+09]];

    PERS robtarget YL61S:=[[0,-102.434,331.364],[0.475779,0.52346,-0.475456,-0.523036],[0,2,0,0],[9E+09,8.10884,48.3912,9E+09,9E+09,9E+09]];
    PERS robtarget YL61E:=[[0,-136.732,324.386],[0.475779,0.52346,-0.475456,-0.523036],[0,2,0,0],[9E+09,8.10884,48.3912,9E+09,9E+09,9E+09]];
    PERS robtarget YL62S:=[[0,-143.638,394.581],[0.461687,0.535407,-0.461915,-0.535556],[0,2,0,0],[9E+09,7.68338,48.3166,9E+09,9E+09,9E+09]];
    PERS robtarget YL62E:=[[0,-165.995,387.902],[0.461687,0.535407,-0.461915,-0.535556],[0,2,0,0],[9E+09,7.68338,48.3166,9E+09,9E+09,9E+09]];
    PERS robtarget YL63S:=[[0,-136.961,363.19],[0.442448,0.551491,-0.442573,-0.551568],[0,2,0,0],[9E+09,9.82577,48.6742,9E+09,9E+09,9E+09]];
    PERS robtarget YL63E:=[[0,-158.994,355.019],[0.442448,0.551491,-0.442573,-0.551568],[0,2,0,0],[9E+09,9.82577,48.6742,9E+09,9E+09,9E+09]];
    PERS robtarget YL67S:=[[0,-100.439,322.029],[0.442448,0.551491,-0.442573,-0.551568],[0,2,0,0],[9E+09,8.96447,48.5355,9E+09,9E+09,9E+09]];
    PERS robtarget YL67E:=[[0.000476837,-134.61,314.453],[0.442448,0.551491,-0.442573,-0.551568],[0,2,0,0],[9E+09,8.96447,48.5355,9E+09,9E+09,9E+09]];
    PERS robtarget YL66S:=[[8,-225,411.8],[0.449728,0.528501,-0.46652,-0.548442],[0,2,0,0],[9E+09,7.65,44.82,9E+09,9E+09,9E+09]];
    PERS robtarget YL66E:=[[8,-189,411.8],[0.449728,0.528501,-0.46652,-0.548442],[0,2,0,0],[9E+09,7.65,44.82,9E+09,9E+09,9E+09]];
    PERS robtarget YL65S:=[[8,-225,411.8],[0.449728,0.528501,-0.46652,-0.548442],[0,2,0,0],[9E+09,7.65,44.82,9E+09,9E+09,9E+09]];
    PERS robtarget YL65E:=[[8,-189,411.8],[0.449728,0.528501,-0.46652,-0.548442],[0,2,0,0],[9E+09,7.65,44.82,9E+09,9E+09,9E+09]];
    PERS robtarget YL64S:=[[8,-225,411.8],[0.449728,0.528501,-0.46652,-0.548442],[0,2,0,0],[9E+09,7.65,44.82,9E+09,9E+09,9E+09]];
    PERS robtarget YL64E:=[[8,-189,411.8],[0.449728,0.528501,-0.46652,-0.548442],[0,2,0,0],[9E+09,7.65,44.82,9E+09,9E+09,9E+09]];
    PERS robtarget YL64KS:=[[0,-236.712,697.465],[0.442448,0.551491,-0.442573,-0.551568],[0,2,0,0],[9E+09,1.26795,46.7321,9E+09,9E+09,9E+09]];
    PERS robtarget YL64KE:=[[0,-260.629,694.325],[0.442448,0.551491,-0.442573,-0.551568],[0,2,0,0],[9E+09,1.26795,46.7321,9E+09,9E+09,9E+09]];
    PERS robtarget YL65KS:=[[0,-226.703,599.049],[0.442448,0.551491,-0.442573,-0.551568],[0,2,0,0],[9E+09,6,48,9E+09,9E+09,9E+09]];
    PERS robtarget YL65KE:=[[0,-249.965,589.663],[0.442448,0.551491,-0.442573,-0.551568],[0,2,0,0],[9E+09,6,48,9E+09,9E+09,9E+09]];
    PERS robtarget YL66KS:=[[0,-204.477,493.494],[0.442448,0.551491,-0.442573,-0.551568],[0,2,0,0],[9E+09,11.127,48.873,9E+09,9E+09,9E+09]];
    PERS robtarget YL66KE:=[[0,-226.433,477.965],[0.442448,0.551491,-0.442573,-0.551568],[0,2,0,0],[9E+09,11.127,48.873,9E+09,9E+09,9E+09]];
    PERS robtarget YL67KS:=[[0,-206.596,501.506],[0.442448,0.551491,-0.442573,-0.551568],[0,2,0,0],[9E+09,10.6921,48.8079,9E+09,9E+09,9E+09]];
    PERS robtarget YL67KE:=[[0,-228.685,486.483],[0.442448,0.551491,-0.442573,-0.551568],[0,2,0,0],[9E+09,10.6921,48.8079,9E+09,9E+09,9E+09]];
    PERS robtarget YL68S:=[[0,-131.055,340.199],[0.428201,0.56264,-0.428263,-0.562735],[0,2,0,0],[9E+09,11.563,48.937,9E+09,9E+09,9E+09]];
    PERS robtarget YL68E:=[[0,-152.782,330.846],[0.428201,0.56264,-0.428263,-0.562735],[0,2,0,0],[9E+09,11.563,48.937,9E+09,9E+09,9E+09]];
    PERS robtarget YL69S:=[[0,-97.8611,310.69],[0.475779,0.52346,-0.475456,-0.523036],[0,2,0,0],[9E+09,9.82577,48.6742,9E+09,9E+09,9E+09]];
    PERS robtarget YL69E:=[[0,-131.894,302.519],[0.475779,0.52346,-0.475456,-0.523036],[0,2,0,0],[9E+09,9.82577,48.6742,9E+09,9E+09,9E+09]];

    PERS robtarget XL69S:=[[141,-57.3,278.76],[0.000117957,0.941052,-0.338263,0.000136519],[0,1,-2,0],[9E+09,9.82577,48.6742,9E+09,9E+09,9E+09]];
    PERS robtarget XL69E:=[[121,-57.3,278.76],[0.000117957,0.941052,-0.338263,0.000136519],[0,1,-2,0],[9E+09,9.82577,48.6742,9E+09,9E+09,9E+09]];
    PERS pose SRL69X:=[[2.79935,-0.0237465,-0.0276489],[1,0,0,0]];

    PERS robtarget XL61S:=[[141,-8.99,-170.4],[0.000212553,0.932221,-0.361891,4.72461E-05],[-1,1,-2,0],[9E+09,8.10884,48.3912,9E+09,9E+09,9E+09]];
    PERS robtarget XL61E:=[[121,-6.78,-73.38],[0.000212323,0.932221,-0.361891,4.67044E-05],[-1,1,-2,0],[9E+09,8.10884,48.3912,9E+09,9E+09,9E+09]];
    PERS pose SRL61X:=[[2.74586,-0.010397,0.00141907],[1,0,0,0]];

    PERS robtarget XL49S:=[[151,-54.59,-184.65],[0.959943,1.46594E-05,7.32901E-06,-0.280197],[-1,1,1,0],[9E+09,-18.2042,49.7958,9E+09,9E+09,9E+09]];
    PERS robtarget XL49E:=[[120.8,-54.59,-184.65],[0.959943,1.46594E-05,7.32901E-06,-0.280197],[-1,1,1,0],[9E+09,-18.2042,49.7958,9E+09,9E+09,9E+09]];
    PERS pose SRL49X:=[[5.36909,-0.00109482,-0.0323181],[1,0,0,0]];

    PERS robtarget YL41air1:=[[356.76,-693.63,1428.70],[0.0565218,0.961931,-0.0569485,0.261249],[-1,0,-2,0],[9E+09,-10.15,44.19,9E+09,9E+09,9E+09]];
    PERS robtarget YL41air2:=[[614.01,-259.36,1104.33],[0.260786,0.144855,-0.889961,-0.344929],[-1,0,0,0],[9E+09,-10.15,44.19,9E+09,9E+09,9E+09]];

    PERS robtarget YL69air1:=[[-261.65,-852.74,1421.82],[0.103662,-0.957671,0.266377,-0.0341167],[-1,0,-1,0],[9E+09,12.53,43.92,9E+09,9E+09,9E+09]];
    PERS robtarget YL69air2:=[[447.24,29.17,714.56],[0.186087,0.688059,-0.699559,-0.0506479],[-1,1,-1,0],[9E+09,12.53,43.92,9E+09,9E+09,9E+09]];

    PERS robtarget XL69air1:=[[268.22,-641.11,985.60],[0.0565186,0.961931,-0.0569466,0.261246],[-1,0,-2,0],[9E+09,-10.15,44.19,9E+09,9E+09,9E+09]];
    PERS robtarget XL69air2:=[[412.80,-348.00,1006.40],[0.0171403,-0.863626,0.502842,-0.031717],[-1,1,-2,0],[9E+09,-10.15,44.19,9E+09,9E+09,9E+09]];
    PERS robtarget XL69air3:=[[241.56,-312.07,489.38],[0.0171461,-0.863629,0.502836,-0.0317137],[-1,1,-2,0],[9E+09,-10.15,44.19,9E+09,9E+09,9E+09]];



    !!!!!!!!!!!!!!!!!!!!!!!!!!!!!!!     M STUFF FOR SIP !!!!!!!!!!!!!!!!!!!!!!!!!!!!!!

!!!!DEFAULT VALUE OF M in the X is -152!!!!!

    PERS robtarget YM41S:=[[-152,-113.919,467.621],[0.587326,-0.393546,-0.587443,0.393802],[-1,1,-3,0],[9E+09,-0.275255,-46.2247,9E+09,9E+09,9E+09]];
    PERS robtarget YM41E:=[[-152,-148.907,468.537],[0.587326,-0.393546,-0.587443,0.393802],[-1,1,-3,0],[9E+09,-0.275255,-46.2247,9E+09,9E+09,9E+09]];

    PERS robtarget YM42S:=[[-152,-110.263,518.104],[0.587415,-0.39386,-0.587303,0.393566],[-1,1,-3,0],[9E+09,-3.95049,-47.5495,9E+09,9E+09,9E+09]];
    PERS robtarget YM42E:=[[-152,-145.038,522.066],[0.587415,-0.39386,-0.587303,0.393566],[-1,1,-3,0],[9E+09,-3.95049,-47.5495,9E+09,9E+09,9E+09]];
    PERS robtarget YM46S:=[[-152,-100.139,577.971],[0.588389,-0.39206,-0.588481,0.392144],[-1,1,-3,0],[9E+09,-8.96447,-48.5355,9E+09,9E+09,9E+09]];
    PERS robtarget YM46E:=[[-152,-134.31,585.547],[0.588389,-0.39206,-0.588481,0.392144],[-1,1,-3,0],[9E+09,-8.96447,-48.5355,9E+09,9E+09,9E+09]];

    PERS robtarget YM45S:=[[-152,-102.234,568.136],[0.588389,-0.392051,-0.588506,0.392117],[-1,1,-3,0],[9E+09,-8.10884,-48.3912,9E+09,9E+09,9E+09]];
    PERS robtarget YM45E:=[[-152,-136.532,575.114],[0.588389,-0.392051,-0.588506,0.392117],[-1,1,-3,0],[9E+09,-8.10884,-48.3912,9E+09,9E+09,9E+09]];
    PERS robtarget YM47S:=[[-152,-90.0267,617.353],[0.560957,-0.430287,-0.561178,0.430418],[-1,1,-3,0],[9E+09,-12.438,-49.062,9E+09,9E+09,9E+09]];
    PERS robtarget YM47E:=[[-152,-123.585,627.294],[0.560868,-0.430402,-0.561091,0.430533],[-1,1,-3,0],[9E+09,-12.438,-49.062,9E+09,9E+09,9E+09]];
    PERS robtarget YM48S:=[[-152,-73.7314,665.293],[0.560884,-0.430683,-0.560804,0.430604],[-1,1,-3,0],[9E+09,-16.8632,-49.6368,9E+09,9E+09,9E+09]];
    PERS robtarget YM48E:=[[-152,-106.296,678.12],[0.560863,-0.430712,-0.560781,0.430633],[-1,1,-3,0],[9E+09,-16.8632,-49.6368,9E+09,9E+09,9E+09]];
    PERS robtarget YM49S:=[[-152,-66.5915,682.424],[0.560794,-0.430638,-0.560829,0.430735],[-1,1,-3,0],[9E+09,-18.2042,-49.7958,9E+09,9E+09,9E+09]];
    PERS robtarget YM49E:=[[-152,-98.8091,696.099],[0.560988,-0.430385,-0.561025,0.43048],[-1,1,-3,0],[9E+09,-18.2042,-49.7958,9E+09,9E+09,9E+09]];


